# B&R Automation Studio project Panasonic_LinkaPowerCP2_A2021055 (part 33)

#### Main.st - Init, cyclic, exit code
```iecst
PROGRAM _INIT

	//Init parametre serva zdvihu výťahu//
	P4_Vytah.ServoZdvihuVytahu.Parameters.Override:= 100;
	P4_Vytah.PAR.Zdvih_JoggRychlost:= 5;
	P4_Vytah.ServoZdvihuVytahu.Command.TorqueLimitation:= TRUE;
	P4_Vytah.ServoZdvihuVytahu.Parameters.Torque:= 1.0;

END_PROGRAM

PROGRAM _CYCLIC

	//Volanie podprogramov a knižníc//
	IOLinkKomunikacia;

	//Volanie funkcie SequenceControl//
	SequenceControl(SC:= SC_P4_Vytah);

	//Enable serva//
	IF Safety.STAV.P4_ZonaVytahu_AKTIVNA AND NOT P4_Vytah.ServoZdvihuVytahu.Command.ErrReset THEN
		P4_Vytah.ServoZdvihuVytahu.Command.PowerON:= TRUE;
	ELSE
		P4_Vytah.ServoZdvihuVytahu.Command.PowerON:= FALSE;
	END_IF

	//Zaokrúhlenie aktuálnej pozície serva zdvihu//
	ServoZdvihu_AktualPosition_UDINT:= REAL_TO_UDINT(P4_Vytah.ServoZdvihuVytahu.Status.ActPosition);

	//Reset poruchy serva//
	IF EDGEPOS(Safety.STAV.P4_ZonaVytahu_AKTIVNA)THEN
		P4_Vytah.ServoZdvihuVytahu.Command.ErrReset:= TRUE;
	END_IF

	CasResetServo_1.IN:= P4_Vytah.ServoZdvihuVytahu.Command.ErrReset;
	IF CasResetServo_1.Q AND NOT P4_Vytah.ServoZdvihuVytahu.Status.Error THEN
		P4_Vytah.ServoZdvihuVytahu.Command.ErrReset:= FALSE;
	END_IF

	CasResetServo_1.PT:= T#500ms;
	CasResetServo_1();

	//Zhasnutie Bannera//
	IF P4_Vytah.CMD.Banner_LED_OFF THEN
		P4_Vytah.Banner.IN.ModraLED_ON:= FALSE;
		P4_Vytah.Banner.IN.CervenaLED_ON:= FALSE;
		P4_Vytah.Banner.IN.CyanLED_ON:= FALSE;
		P4_Vytah.Banner.IN.ModraRotujucaLED_ON:= FALSE;
		P4_Vytah.Banner.IN.OranzovaLED_ON:= FALSE;
		P4_Vytah.Banner.IN.ZelenaLED_ON:= FALSE;
		P4_Vytah.Banner.IN.ZltaLED_ON:= FALSE;
		P4_Vytah.CMD.Banner_LED_OFF:= FALSE;
	END_IF

	//Reset sekcie //
	IF P4_Vytah.Reset THEN
		SC_P4_Vytah.Step:= 0;
		P4_Vytah.ServoZdvihuVytahu.Command.ErrReset:= TRUE;
		P4_Vytah.Reset:= FALSE;
	ELSIF NOT Safety.STAV.Linka_ZonaCS_AKTIVNA THEN
		SC_P4_Vytah.Step:= 0;
	END_IF

	CASE SC_P4_Vytah.Step OF

		0:
			SC_P4_Vytah.StepName:='0 - Nulovanie';
			P4_Vytah.Automat:= FALSE;
			P4_Vytah.KoniecCyklu:= FALSE;
			P4_Vytah.Manual:= FALSE;
			P4_Vytah.STAV.PoINIT:= FALSE;
			P4_Vytah.ServoZdvihuVytahu.Command.JogNeg:= FALSE;
			P4_Vytah.ServoZdvihuVytahu.Command.JogPos:= FALSE;
			P4_Vytah.ServoZdvihuVytahu.Command.MoveAdditive:= FALSE;
			P4_Vytah.ServoZdvihuVytahu.Command.MovePosition:= FALSE;
			IF NOT P4_Vytah.ServoZdvihuVytahu.Status.StandStill THEN
				P4_Vytah.ServoZdvihuVytahu.Command.Stop:= TRUE;
			END_IF
			P4_Vytah.OUT.DopravnikChod_VPRED:= FALSE;
			P4_Vytah.OUT.DopravnikChod_VZAD:= FALSE;
			P4_Vytah.CMD.Banner_LED_OFF:= TRUE;
			P4_Vytah.RFID_hlava.PrecitajChipRFID:= FALSE;
			TRCB_P4_Vytah_ST10.CMD.VyziadajStavPaletky_TYP1:= FALSE;
			TRCB_P4_Vytah_ST10.CMD.PriradQRkodFiltra_TYP3:= FALSE;
			TRCB_P4_Vytah_ST10.CMD.OdosliStavPaletky_TYP2:= FALSE;
			TRCB_P4_Vytah_ST10.CMD.VyziadajStavPanatrace_TYP4:= FALSE;
			P4_Vytah.CMD.RR_ChodDopravnika_VPRED:= FALSE;
			P4_Vytah.CMD.RR_ChodDopravnika_VZAD:= FALSE;
			P4_Vytah.CMD.RR_ZdvihVytahu_DOLE:= FALSE;
			P4_Vytah.CMD.RR_ZdvihVytahu_HORE:= FALSE;
			CAM16.CMD.Triger:= FALSE;
			CAM16.STAV.Results_READY:= FALSE;
			FTP_CAM16.CMD.OdosliFotku:= FALSE;
			FTP_CAM16.CMD.VymazFotku:= FALSE;
			P34_Vizu.ZobrazHL1_ST10:= FALSE;
			P34_Vizu.ZobrazHL2_ST10:= FALSE;
			P34_Vizu.ZobrazHL3_ST10:= FALSE;
			P34_Vizu.ZobrazHL4_ST10:= FALSE;
			P34_Vizu.ZobrazHL5_ST10:= FALSE;
			P34_Vizu.ZobrazHL6_ST10:= FALSE;
			P34_Vizu.ZobrazHL7_ST10:= FALSE;
			P34_Vizu.ZobrazHL8_ST10:= FALSE;
			P34_Vizu.ZobrazHL9_ST10:= FALSE;
			P34_Vizu.ZobrazHL10_ST10:= FALSE;
			P4_Vytah_KAM_Result_Ignoruj:= FALSE;
			P4_Vytah_KAM_Result_OK:= FALSE;
			P4_Vytah_KAM_Result_NG:= FALSE;
			P4_Vytah.PAR.IndexFotky:= 0;
			TRCB_P4_Vytah_OpatovnyDopyt:= FALSE;
			TRCB_P4_Vytah_PaletkaNG:= FALSE;
			PocetTrigrovKamery:= 0;
			PocetDopytovNaServer:= 0;
			CisloFotky:= 0;
			TestovaciKus:= FALSE;
			Stav_VlozenaPaletka:= FALSE;
			P4_Vytah_Taktime.IN.START_MeraniaCasu:= FALSE;
			P4_Etiketovacka.STAV.PrebiehaVyvezeniePaletky:= FALSE;
			P4_Vytah.STAV.PrebiehaVyvezeniePaletky:= FALSE;
			P4_Vytah_Taktime.IN.START_MeraniaStratovehoCasu:= FALSE;

			IF Safety.STAV.P4_ZonaVytahu_AKTIVNA AND
				P4_Pracovisko.STAV.HardwareVytahu_OK AND
				NOT P4_Pracovisko.STAV.Porucha_ST6 AND
				(P4_Vytah.ServoZdvihuVytahu.Status.Ready AND P4_Vytah.ServoZdvihuVytahu.Status.StandStill) THEN
				P4_Vytah.ServoZdvihuVytahu.Command.Stop:= FALSE;
				SC_P4_Vytah.ResetStep:= TRUE;
				SC_P4_Vytah.Step:= 1;
			END_IF

		1:
			SC_P4_Vytah.StepName:='1 - Cakam na spustenie vyroby';
			P4_Vytah.KoniecCyklu:= FALSE;
			IF P4_Vytah.Automat THEN
				SC_P4_Vytah.Step:= 2;
			ELSIF P4_Vytah.Manual THEN
				SC_P4_Vytah.Step:= 700;
			END_IF

			//********************************************************Inicializácia****************************************************************************//

		2:
			SC_P4_Vytah.StepName:='2 - Inicializacia - cakam na spustenie inicializacie';
			SC_P4_Vytah.IdleTime.PT:= T#2s;
			SC_P4_Vytah.AlarmTime.PT:= T#5s;

			SC_P4_Vytah.IdleTime.IN:= P4_Dopravniky.STAV.PoINIT;

			P4_Vytah.ServoZdvihuVytahu.Parameters.Acc:= P34_RemPremenne.P4_Vytah_Zdvih_Acc;
			P4_Vytah.ServoZdvihuVytahu.Parameters.Dcc:= P34_RemPremenne.P4_Vytah_Zdvih_Dcc;
			P4_Vytah.ServoZdvihuVytahu.Parameters.Torque:= 1.5;

			IF SC_P4_Vytah.IdleTime.Q THEN
				SC_P4_Vytah.ResetStep:= TRUE;
				SC_P4_Vytah.Step:= 3;
			END_IF

		3:
			SC_P4_Vytah.StepName:='3 - Inicializacia - vymazanie adresara kamery';
			SC_P4_Vytah.IdleTime.PT:= T#4s;
			SC_P4_Vytah.AlarmTime.PT:= T#5s;

			P4_Vytah.Banner.IN.ModraLED_ON:= TRUE;

			IF NOT SC_P4_Vytah.Switch1 THEN
				FTP_CAM16.CMD.VymazFotku:= TRUE;
				SC_P4_Vytah.Switch1:= TRUE;
			END_IF

			IF FTP_CAM16.STATUS.KomunikaciaUkoncena THEN
				P4_Vytah.CMD.Banner_LED_OFF:= TRUE;
				FTP_CAM16.CMD.VymazFotku:= FALSE;
				SC_P4_Vytah.ResetStep:= TRUE;
				SC_P4_Vytah.Step:= 4;
			ELSIF FTP_CAM16.STATUS.KomunikaciaError THEN
				P34_Alarmy[410]:= TRUE;
				P4_Pracovisko.STAV.Porucha_ST6:= TRUE;
			END_IF

		4:
			SC_P4_Vytah.StepName:='4 - Inicializacia - spustam dopravnik vytahu pre navezenie paletky';
			SC_P4_Vytah.IdleTime.PT:= T#500ms;
			SC_P4_Vytah.AlarmTime.PT:= T#7s;

			SC_P4_Vytah.IdleTime.IN:= P4_Vytah.RFID_hlava.PritomnostPaletky;

			IF NOT SC_P4_Vytah.Switch1 THEN
				P4_Vytah.OUT.DopravnikChod_VPRED:= TRUE;
				SC_P4_Vytah.AlarmTime.IN:= TRUE;
				SC_P4_Vytah.Switch1:= TRUE;
			END_IF

			IF SC_P4_Vytah.IdleTime.Q AND NOT P4_Vytah.IN.PrechodDopravnika THEN
				P4_Vytah.OUT.DopravnikChod_VPRED:= FALSE;
				SC_P4_Vytah.ResetStep:= TRUE;
				SC_P4_Vytah.Step:= 13;
			ELSIF SC_P4_Vytah.AlarmTime.Q AND NOT P4_Vytah.RFID_hlava.PritomnostPaletky AND NOT P4_Vytah.IN.PrechodDopravnika THEN
				P4_Vytah.OUT.DopravnikChod_VPRED:= FALSE;
				SC_P4_Vytah.ResetStep:= TRUE;
				SC_P4_Vytah.Step:= 13;
			ELSIF SC_P4_Vytah.IdleTime.Q AND P4_Vytah.IN.PrechodDopravnika THEN
				P34_Alarmy[411]:= TRUE;
				P4_Pracovisko.STAV.Porucha_ST6:= TRUE;
			END_IF

		13:
			SC_P4_Vytah.StepName:='13 - Inicializacia - presuvam vytah do hornej pozicie vyvazania';
			SC_P4_Vytah.IdleTime.PT:= T#1s;
			SC_P4_Vytah.AlarmTime.PT:= T#5s;

			SC_P4_Vytah.IdleTime.IN:= Safety.STAV.P4_Vytah_Bariera_AKTIVNA;
			P34_Vizu.ZobrazHL6_ST10:= NOT Safety.STAV.P4_Vytah_Bariera_AKTIVNA;

			P4_Vytah.ServoZdvihuVytahu.Parameters.Velocity:= P34_RemPremenne.P4_Vytah_RychlostZdvihu/1000;
			P4_Vytah.ServoZdvihuVytahu.Parameters.Position:= P34_RemPremenne.P4_Vytah_PoziciaNakladania;

			P4_Vytah.Banner.IN.OranzovaLED_ON:= Blikac1s;

			IF NOT SC_P4_Vytah.Switch1 AND SC_P4_Vytah.IdleTime.Q THEN
				P4_Vytah.ServoZdvihuVytahu.Command.MovePosition:= TRUE;
				SC_P4_Vytah.Switch1:= TRUE;
			END_IF

			IF EDGEPOS(P4_Vytah.ServoZdvihuVytahu.Status.InPosition) THEN
				P4_Vytah.ServoZdvihuVytahu.Command.MovePosition:= FALSE;
				P4_Vytah.CMD.Banner_LED_OFF:= TRUE;
				P34_Vizu.ZobrazHL6_ST10:= FALSE;
				SC_P4_Vytah.ResetStep:= TRUE;
				SC_P4_Vytah.Step:= 15;
			END_IF

		15:
			SC_P4_Vytah.StepName:='15 - Inicializacia - kontrola pritomnosti paletky';
			SC_P4_Vytah.IdleTime.PT:= T#2s;
			SC_P4_Vytah.AlarmTime.PT:= T#5s;

			IF P4_Vytah.RFID_hlava.PritomnostPaletky THEN
				SC_P4_Vytah.ResetStep:= TRUE;
				SC_P4_Vytah.Step:= 18;
			ELSE
				P4_Vytah.STAV.PoINIT:= TRUE;
				SC_P4_Vytah.ResetStep:= TRUE;
				SC_P4_Vytah.Step:= 100;
			END_IF

		18:
			SC_P4_Vytah.StepName:='18 - Inicializacia -  precitanie cisla paletky';
			SC_P4_Vytah.IdleTime.PT:= T#200ms;
			SC_P4_Vytah.AlarmTime.PT:= T#5s;

			SC_P4_Vytah.IdleTime.IN:= P4_Vytah.RFID_hlava.PritomnostPaletky;

			IF SC_P4_Vytah.IdleTime.Q AND NOT SC_P4_Vytah.Switch1 THEN
				P4_Vytah.RFID_hlava.PrecitajChipRFID:= TRUE;
				i:= 0;
				SC_P4_Vytah.Switch1:= TRUE;
			END_IF

			IF P4_Vytah.RFID_hlava.Stav_CitanieZapis_OK AND P4_Vytah.RFID_hlava.PrecitaneCisloPaletky <> 0 THEN
				i:= P4_Vytah.RFID_hlava.PrecitaneCisloPaletky;
				P4_Vytah.PAR.CisloPaletky:= P4_Vytah.RFID_hlava.PrecitaneCisloPaletky;
				P4_Vytah.RFID_hlava.PrecitajChipRFID:= FALSE;
				SC_P4_Vytah.ResetStep:= TRUE;
				SC_P4_Vytah.Step:= 20;
			END_IF

		20:
			SC_P4_Vytah.StepName:='20 - Inicializacia - priradenie indexu paletky na zaklade precitanej hodnoty';
			SC_P4_Vytah.IdleTime.PT:= T#200ms;
			SC_P4_Vytah.AlarmTime.PT:= T#5s;

			IF i<> 0 THEN
				P4_Vytah.PAR.CisloPaletky_STRING:= USINT_TO_STRING(i);
				Paletka[i].PAR.CisloPaletky:= USINT_TO_STRING(i);
				SC_P4_Vytah.ResetStep:= TRUE;
				SC_P4_Vytah.Step:= 30;
			ELSE
				P34_Alarmy[418]:= TRUE;
				P4_Pracovisko.STAV.Porucha_ST6:= TRUE;
			END_IF

		30:
			SC_P1_StoperSrobovania.StepName:='30 - Inicializacia - kontrola stavu paletky';
			SC_P4_Vytah.IdleTime.PT:= T#200ms;
			SC_P4_Vytah.AlarmTime.PT:= T#5s;

			IF Paletka[i].STAV.StavPaletky = '' THEN
				P4_Vytah.STAV.PoINIT:= TRUE;
				Paletka[i].STAV.StavPaletky:= 'NG';
				SC_P4_Vytah.ResetStep:= TRUE;
				SC_P4_Vytah.Step:= 560;
			ELSIF Paletka[i].STAV.StavPaletky = 'PRECH' THEN
				P4_Vytah.STAV.PoINIT:= TRUE;
				SC_P4_Vytah.ResetStep:= TRUE;
				SC_P4_Vytah.Step:= 130;
			ELSIF Paletka[i].STAV.StavPaletky = 'TEST' THEN
				P4_Vytah.STAV.PoINIT:= TRUE;
				SC_P4_Vytah.ResetStep:= TRUE;
				SC_P4_Vytah.Step:= 130;
			ELSIF Paletka[i].STAV.StavPaletky = 'REV' AND Paletka[i].STAV.CisloRevorkovejStanice = 'ST_10' THEN
				Paletka[i].STAV.StavPaletky:= 'OK';
				SC_P4_Vytah.ResetStep:= TRUE;
				SC_P4_Vytah.Step:= 33;
			ELSIF Paletka[i].STAV.StavPaletky = 'REV' AND Paletka[i].STAV.CisloRevorkovejStanice <> 'ST_10' THEN
				P4_Vytah.STAV.PoINIT:= TRUE;
				SC_P4_Vytah.ResetStep:= TRUE;
				SC_P4_Vytah.Step:= 130;
			ELSIF Paletka[i].STAV.StavPaletky = 'OK' THEN
				SC_P4_Vytah.ResetStep:= TRUE;
				SC_P4_Vytah.Step:= 33;
			ELSIF Paletka[i].STAV.StavPaletky = 'NG' THEN
				P4_Vytah.STAV.PoINIT:= TRUE;
				SC_P4_Vytah.ResetStep:= TRUE;
				SC_P4_Vytah.Step:= 130;
			END_IF

		33:
			SC_P4_Vytah.StepName:='33 - Inicializacia - kontrola uzavretia komunikacie s Panatrace';
			SC_P4_Vytah.IdleTime.PT:= T#5s;
			SC_P4_Vytah.AlarmTime.PT:= T#5s;

			IF Paletka[i].STAV.Komunikacia_DONE THEN
				P4_Vytah.STAV.PoINIT:= TRUE;
				SC_P4_Vytah.ResetStep:= TRUE;
				SC_P4_Vytah.Step:= 130;
			ELSE
				P4_Vytah.STAV.PoINIT:= TRUE;
				SC_P4_Vytah.ResetStep:= TRUE;
				SC_P4_Vytah.Step:= 111;
			END_IF

			//********************************************************Automatický režim****************************************************************************//

		100:
			SC_P4_Vytah.StepName:='100 - Automaticky Rezim - cakam na navezenie paletky na vytah z vrchneho dopravnika';
			SC_P4_Vytah.IdleTime.PT:= T#200ms;
			SC_P4_Vytah.AlarmTime.PT:= T#5s;

			P4_Vytah.ServoZdvihuVytahu.Parameters.Acc:= P34_RemPremenne.P4_Vytah_Zdvih_Acc;
			P4_Vytah.ServoZdvihuVytahu.Parameters.Dcc:= P34_RemPremenne.P4_Vytah_Zdvih_Dcc;
			P4_Vytah.ServoZdvihuVytahu.Parameters.Torque:= 1.5;

			IF P4_Vytah.KoniecCyklu AND NOT P4_Etiketovacka.Automat THEN
				SC_P4_Vytah.ResetStep:= TRUE;
				SC_P4_Vytah.Step:= 0;
			ELSIF SC_P4_Etiketovacka.Step = 561 AND NOT P4_Vytah.RFID_hlava.PritomnostPaletky AND NOT P4_Vytah.IN.PrechodDopravnika THEN
				Stav_VlozenaPaletka:= FALSE;
				SC_P4_Vytah.ResetStep:= TRUE;
				SC_P4_Vytah.Step:= 101;
			ELSIF P4_Vytah.RFID_hlava.PritomnostPaletky THEN
				P4_Etiketovacka.STAV.PrebiehaVyvezeniePaletky:= FALSE;
				Stav_VlozenaPaletka:= TRUE;
				SC_P4_Vytah.ResetStep:= TRUE;
				SC_P4_Vytah.Step:= 105;
			END_IF

		101:
			SC_P4_Vytah.StepName:='101 - Automaticky Rezim - navazam paletku na dopravnik vytahu';
			SC_P4_Vytah.IdleTime.PT:= T#200ms;
			SC_P4_Vytah.AlarmTime.PT:= T#20s;

			SC_P4_Vytah.IdleTime.IN:= P4_Vytah.RFID_hlava.PritomnostPaletky;

			IF NOT SC_P4_Vytah.Switch2 AND P4_Vytah.RFID_hlava.PritomnostPaletky THEN
				P4_Vytah_Taktime.IN.START_MeraniaCasu:= TRUE;
				P4_Vytah_Taktime.IN.ZAPIS_MeraniaCasu:= TRUE;
				P4_Vytah_Taktime.IN.ZAPIS_StratovyCas:= TRUE;
				Buffer_14.Hodnota:= P4_Vytah_Taktime.OUT.StratoveSekundy;
				Buffer_14.ZapisHodnotu:= TRUE;
				SC_P4_Vytah.Switch2:= TRUE;
			END_IF

			IF NOT SC_P4_Vytah.Switch1 THEN
				P4_Vytah.OUT.DopravnikChod_VPRED:= TRUE;
				SC_P4_Vytah.AlarmTime.IN:= TRUE;
				SC_P4_Vytah.Switch1:= TRUE;
			END_IF

			IF SC_P4_Vytah.IdleTime.Q THEN
				P4_Etiketovacka.STAV.PrebiehaVyvezeniePaletky:= FALSE;
				P4_Vytah.OUT.DopravnikChod_VPRED:= FALSE;
				SC_P4_Vytah.ResetStep:= TRUE;
				SC_P4_Vytah.Step:= 105;
			ELSIF SC_P4_Vytah.AlarmTime.Q THEN
				P34_Alarmy[416]:= TRUE;
				P4_Pracovisko.STAV.Porucha_ST6:= TRUE;
			END_IF

		105:
			SC_P4_Vytah.StepName:='105 - Automaticky Rezim - precitanie cisla paletky';
			SC_P4_Vytah.IdleTime.PT:= T#500ms;
			SC_P4_Vytah.AlarmTime.PT:= T#5s;
			SC_P4_Vytah.IdleTime.IN:= TRUE;

			IF NOT SC_P4_Vytah.Switch1 THEN
				i:= 0;
				P4_Vytah.RFID_hlava.PrecitajChipRFID:= TRUE;
				SC_P4_Vytah.Switch1:= TRUE;
			END_IF

			IF P4_Vytah.RFID_hlava.Stav_CitanieZapis_OK AND P4_Vytah.RFID_hlava.PrecitaneCisloPaletky <> 0 THEN
				i:= P4_Vytah.RFID_hlava.PrecitaneCisloPaletky;
				P4_Vytah.PAR.CisloPaletky:= P4_Vytah.RFID_hlava.PrecitaneCisloPaletky;
				P4_Vytah.RFID_hlava.PrecitajChipRFID:= FALSE;
				SC_P4_Vytah.ResetStep:= TRUE;
				SC_P4_Vytah.Step:= 108;
			END_IF

		108:
			SC_P4_Vytah.StepName:='108 - Automaticky Rezim - kontrola a priradenie indexu paletky na zaklade precitanej hodnoty';
			SC_P4_Vytah.IdleTime.PT:= T#200ms;
			SC_P4_Vytah.AlarmTime.PT:= T#5s;

			IF i<> 0 THEN
				P4_Vytah.PAR.CisloPaletky_STRING:= USINT_TO_STRING(i);
				Paletka[i].PAR.CisloPaletky:= USINT_TO_STRING(i);
				SC_P4_Vytah.ResetStep:= TRUE;
				SC_P4_Vytah.Step:= 110;
			ELSE
				P34_Alarmy[418]:= TRUE;
				P4_Pracovisko.STAV.Porucha_ST6:= TRUE;
			END_IF

		110:
			SC_P4_Vytah.StepName:='110 - Automaticky Rezim - kontrola stavu paletky';
			SC_P4_Vytah.IdleTime.PT:= T#200ms;
			SC_P4_Vytah.AlarmTime.PT:= T#5s;

			IF Paletka[i].STAV.StavPaletky = '' THEN
				Paletka[i].STAV.StavPaletky:= 'NG';
				SC_P4_Vytah.ResetStep:= TRUE;
				SC_P4_Vytah.Step:= 560;
			ELSIF Paletka[i].STAV.StavPaletky = 'PRECH' THEN
				SC_P4_Vytah.ResetStep:= TRUE;
				SC_P4_Vytah.Step:= 130;
			ELSIF Paletka[i].STAV.StavPaletky = 'TEST' THEN
				SC_P4_Vytah.ResetStep:= TRUE;
				SC_P4_Vytah.Step:= 130;
			ELSIF Paletka[i].STAV.StavPaletky = 'REV' AND Paletka[i].STAV.CisloRevorkovejStanice = 'ST_10' THEN
				Paletka[i].STAV.StavPaletky:= 'OK';
				SC_P4_Vytah.ResetStep:= TRUE;
				SC_P4_Vytah.Step:= 111;
			ELSIF Paletka[i].STAV.StavPaletky = 'REV' AND Paletka[i].STAV.CisloRevorkovejStanice <> 'ST_10' THEN
				SC_P4_Vytah.ResetStep:= TRUE;
				SC_P4_Vytah.Step:= 130;
			ELSIF Paletka[i].STAV.StavPaletky = 'OK' THEN
				SC_P4_Vytah.ResetStep:= TRUE;
				SC_P4_Vytah.Step:= 111;
			ELSIF Paletka[i].STAV.StavPaletky = 'NG' THEN
				SC_P4_Vytah.ResetStep:= TRUE;
				SC_P4_Vytah.Step:= 130;
			END_IF

		111:
			SC_P4_Vytah.StepName:='111 - Automaticky Rezim - kontrola prihlasenia operatora';
			SC_P4_Vytah.IdleTime.PT:= T#1s;
			SC_P4_Vytah.AlarmTime.PT:= T#5s;

			IF P34_UzivatelPrihlaseny THEN
				Paletka[i].PAR.ID_Operatora:= 'E2';//UsersVizu.CisloPrihlasenejKarty_Panel3;
				P34_Vizu.ZobrazHL7_ST10:= FALSE;
				P4_Vytah.CMD.Banner_LED_OFF:= FALSE;
				SC_P4_Vytah.ResetStep:= TRUE;
				SC_P4_Vytah.Step:= 112;
			ELSE
				P4_Vytah.Banner.IN.CyanLED_ON:= Blikac500ms;
				P34_Vizu.ZobrazHL7_ST10:= TRUE;
				Paletka[i].PAR.ID_Operatora:= '';
			END_IF

		112:
			SC_P4_Vytah.StepName:='112 - Automaticky Rezim - vyziadanie stavu komunikacie zo serverom';
			SC_P4_Vytah.IdleTime.PT:= T#200ms;
			SC_P4_Vytah.AlarmTime.PT:= T#10s;

			P4_Vytah.Banner.IN.ModraRotujucaLED_ON:= TRUE;

			IF Linka.KOM_Panatrace_OFF THEN
				CAM16.STAV.Results_READY:= FALSE;
				CAM16.STAV.OldRunCounter:= CAM16.STAV.RunCounter;
				P4_Vytah.CMD.Banner_LED_OFF:= TRUE;
				SC_P4_Vytah.ResetStep:= TRUE;
				SC_P4_Vytah.Step:= 118;
			ELSIF NOT SC_P4_Vytah.Switch1 AND TRCB_P4_Vytah_ST10.STATUS.KOM_READY THEN
				TRCB_P4_Vytah_ST10.CMD.VyziadajStavPanatrace_TYP4:= TRUE;
				(*P4_Vytah_Taktime.IN.START_MeraniaStratovehoCasu:= TRUE;*)
				SC_P4_Vytah.Switch1:= TRUE;
			END_IF

			IF TRCB_P4_Vytah_ST10.STATUS.KomunikaciaUkoncena THEN
				P4_Vytah.CMD.Banner_LED_OFF:= TRUE;
				TRCB_P4_Vytah_ST10.CMD.VyziadajStavPanatrace_TYP4:= FALSE;
				P4_Vytah_Taktime.IN.START_MeraniaStratovehoCasu:= FALSE;
				SC_P4_Vytah.ResetStep:= TRUE;
				SC_P4_Vytah.Step:= 113;
			ELSIF TRCB_P4_Vytah_ST10.STATUS.KomunikaciaError THEN
				P4_Vytah.CMD.Banner_LED_OFF:= TRUE;
				TRCB_P4_Vytah_ST10.CMD.VyziadajStavPanatrace_TYP4:= FALSE;
				P4_Vytah_Taktime.IN.START_MeraniaStratovehoCasu:= FALSE;
				SC_P4_Vytah.ResetStep:= TRUE;
				SC_P4_Vytah.Step:= 114;
			END_IF

		113:
			SC_P4_Vytah.StepName:='113 - Automaticky Rezim - kontrola odpovede servera';
			SC_P4_Vytah.IdleTime.PT:= T#200ms;
			SC_P4_Vytah.AlarmTime.PT:= T#5s;

			IF NOT TRCB_P4_Vytah_ST10.STATUS.KomunikaciaUkoncena THEN
				IF TRCB_P4_Vytah_ST10.OUTPUTS.DruhCinnostiNaPaletke = '0;Generating' THEN
					SC_P4_Vytah.ResetStep:= TRUE;
					SC_P4_Vytah.Step:= 114;
				ELSIF TRCB_P4_Vytah_ST10.OUTPUTS.DruhCinnostiNaPaletke = '1;Request' THEN
					SC_P4_Vytah.ResetStep:= TRUE;
					SC_P4_Vytah.Step:= 115;
				ELSIF TRCB_P4_Vytah_ST10.OUTPUTS.DruhCinnostiNaPaletke = '2;Report' THEN
					CAM16.STAV.OldRunCounter:= CAM16.STAV.RunCounter;
					CAM16.STAV.Results_READY:= FALSE;
					SC_P4_Vytah.ResetStep:= TRUE;
					SC_P4_Vytah.Step:= 118;
				ELSIF TRCB_P4_Vytah_ST10.OUTPUTS.DruhCinnostiNaPaletke = '3;Wedding' THEN
					SC_P4_Vytah.ResetStep:= TRUE;
					SC_P4_Vytah.Step:= 114;
				ELSIF TRCB_P4_Vytah_ST10.OUTPUTS.DruhCinnostiNaPaletke = '4;Status' THEN
					SC_P4_Vytah.ResetStep:= TRUE;
					SC_P4_Vytah.Step:= 114;
				ELSIF TRCB_P4_Vytah_ST10.OUTPUTS.DruhCinnostiNaPaletke = '5;' THEN
					SC_P4_Vytah.ResetStep:= TRUE;
					SC_P4_Vytah.Step:= 114;
				ELSE
					SC_P4_Vytah.ResetStep:= TRUE;
					SC_P4_Vytah.Step:= 114;
				END_IF
			END_IF

		114:
			SC_P4_Vytah.StepName:='114 - Automaticky Rezim - rozhodnutie obsluhy po chybe komunikacie s Panatrace';
			SC_P4_Vytah.IdleTime.PT:= T#200ms;
			SC_P4_Vytah.AlarmTime.PT:= T#5s;

			P34_Vizu.ZobrazHL10_ST10:= TRUE;

			IF TRCB_P4_Vytah_OpatovnyDopyt THEN
				TRCB_P4_Vytah_OpatovnyDopyt:= FALSE;
				P34_Vizu.ZobrazHL10_ST10:= FALSE;
				SC_P4_Vytah.ResetStep:= TRUE;
				SC_P4_Vytah.Step:= 112;
			ELSIF TRCB_P4_Vytah_PaletkaNG THEN
				TRCB_P4_Vytah_PaletkaNG:= FALSE;
				P34_Vizu.ZobrazHL10_ST10:= FALSE;
				Paletka[i].STAV.StavPaletky := 'NG';
				SC_P4_Vytah.ResetStep:= TRUE;
				SC_P4_Vytah.Step:= 130;
			END_IF

		115:
			SC_P4_Vytah.StepName:='115 - Automaticky Rezim - vyziadanie stavu paletky zo servera';
			SC_P4_Vytah.IdleTime.PT:= T#200ms;
			SC_P4_Vytah.AlarmTime.PT:= T#5s;
			SC_P4_Vytah.IdleTime.IN:= TRUE;

			IF NOT SC_P4_Vytah.Switch1 AND TRCB_P4_Vytah_ST10.STATUS.KOM_READY THEN
				TRCB_P4_Vytah_ST10.CMD.VyziadajStavPaletky_TYP1:= TRUE;
				(*P4_Vytah_Taktime.IN.START_MeraniaStratovehoCasu:= TRUE;*)
				SC_P4_Vytah.Switch1:= TRUE;
			END_IF

			IF TRCB_P4_Vytah_ST10.STATUS.KomunikaciaUkoncena THEN
				P4_Vytah.CMD.Banner_LED_OFF:= TRUE;
				TRCB_P4_Vytah_ST10.CMD.VyziadajStavPaletky_TYP1:= FALSE;
				P4_Vytah_Taktime.IN.START_MeraniaStratovehoCasu:= FALSE;
				SC_P4_Vytah.ResetStep:= TRUE;
				SC_P4_Vytah.Step:= 116;
			ELSIF TRCB_P4_Vytah_ST10.STATUS.KomunikaciaError THEN
				P4_Vytah.CMD.Banner_LED_OFF:= TRUE;
				TRCB_P4_Vytah_ST10.CMD.VyziadajStavPaletky_TYP1:= FALSE;
				P4_Vytah_Taktime.IN.START_MeraniaStratovehoCasu:= FALSE;
				SC_P4_Vytah.ResetStep:= TRUE;
				SC_P4_Vytah.Step:= 114;
			END_IF

		116:
			SC_P4_Vytah.StepName:='116 - Automaticky Rezim - kontrola odpovede servera';
			SC_P4_Vytah.IdleTime.PT:= T#200ms;
			SC_P4_Vytah.AlarmTime.PT:= T#5s;

			IF NOT TRCB_P4_Vytah_ST10.STATUS.KomunikaciaUkoncena THEN
				IF TRCB_P4_Vytah_ST10.OUTPUTS.PovolenieCinnostiNaPaletke = 'OK' THEN
					CAM16.STAV.Results_READY:= FALSE;
					CAM16.STAV.OldRunCounter:= CAM16.STAV.RunCounter;
					SC_P4_Vytah.ResetStep:= TRUE;
					SC_P4_Vytah.Step:= 118;
				ELSIF TRCB_P4_Vytah_ST10.OUTPUTS.PovolenieCinnostiNaPaletke = 'NG' THEN
					SC_P4_Vytah.ResetStep:= TRUE;
					SC_P4_Vytah.Step:= 117;
				END_IF
			END_IF

		117:
			SC_P4_Vytah.StepName:='117 - Automaticky Rezim - rozhodnutie obsluhy po odpovedi panatrace NG';
			SC_P4_Vytah.IdleTime.PT:= T#200ms;
			SC_P4_Vytah.AlarmTime.PT:= T#5s;

			P34_Vizu.ZobrazHL9_ST10:= TRUE;

			IF TRCB_P4_Vytah_OpatovnyDopyt THEN
				TRCB_P4_Vytah_OpatovnyDopyt:= FALSE;
				P34_Vizu.ZobrazHL9_ST10:= FALSE;
				SC_P4_Vytah.ResetStep:= TRUE;
				SC_P4_Vytah.Step:= 112;
			ELSIF TRCB_P4_Vytah_PaletkaNG THEN
				TRCB_P4_Vytah_PaletkaNG:= FALSE;
				P34_Vizu.ZobrazHL9_ST10:= FALSE;
				Paletka[i].STAV.StavPaletky := 'NG';
				SC_P4_Vytah.ResetStep:= TRUE;
				SC_P4_Vytah.Step:= 130;
			END_IF

		118:
			SC_P4_Vytah.StepName:='118 - Automaticky Rezim - kamerova kontrola paletky CAM16';//CAM 16
			SC_P4_Vytah.IdleTime.PT:= T#5s;
			SC_P4_Vytah.AlarmTime.PT:= T#5s;

			P4_Vytah.Banner.IN.ModraLED_ON:= TRUE;

			IF NOT SC_P4_Vytah.Switch1 AND CAM16.STAV.Command_READY THEN
				CAM16.CMD.Triger:= TRUE;
				SC_P4_Vytah.IdleTime.IN:= TRUE;
				SC_P4_Vytah.Switch1:= TRUE;
			END_IF

			IF CAM16.STAV.Results_READY AND CAM16.STAV.Command_AKCEPTOVANY AND CAM16.STAV.OldRunCounter <> CAM16.STAV.RunCounter THEN
				PocetTrigrovKamery:= 0;
				CAM16.STAV.Results_READY:= FALSE;
				CAM16.STAV.OldRunCounter:= CAM16.STAV.RunCounter;
				CAM16.CMD.Triger:= FALSE;
				P4_Vytah.CMD.Banner_LED_OFF:= TRUE;
				SC_P4_Vytah.ResetStep:= TRUE;
				SC_P4_Vytah.Step:= 120;
			ELSIF SC_P4_Vytah.IdleTime.Q AND PocetTrigrovKamery < 5 THEN
				PocetTrigrovKamery:= PocetTrigrovKamery + 1;
				CAM16.CMD.Triger:= FALSE;
				CAM16.STAV.Results_READY:= FALSE;
				CAM16.STAV.OldRunCounter:= CAM16.STAV.RunCounter;
				P4_Vytah.CMD.Banner_LED_OFF:= TRUE;
				SC_P4_Vytah.ResetStep:= TRUE;
				SC_P4_Vytah.Step:= 119;
			ELSIF SC_P4_Vytah.IdleTime.Q AND PocetTrigrovKamery >= 5 THEN
				P34_Alarmy[455]:= TRUE;
				P4_Pracovisko.STAV.Porucha_ST6:= TRUE;
			END_IF

		119:
			SC_P4_Vytah.StepName:='119 - Automaticky Rezim - cakam na opatovny triger kamery CAM16';
			SC_P4_Vytah.IdleTime.PT:= T#1s;
			SC_P4_Vytah.AlarmTime.PT:= T#5s;

			SC_P4_Vytah.IdleTime.IN:= TRUE;

			IF SC_P4_Vytah.IdleTime.Q THEN
				SC_P4_Vytah.ResetStep:= TRUE;
				SC_P4_Vytah.Step:= 118;
			END_IF

		120:
			SC_P4_Vytah.StepName:='120 - Automaticky Rezim - vysledok kamerovej kontroly kamery CAM16';
			SC_P4_Vytah.IdleTime.PT:= T#1s;
			SC_P4_Vytah.AlarmTime.PT:= T#5s;

			IF Linka.P4_Kamery_OFF THEN
				CAM16.CMD.Triger:= FALSE;
				CAM16.PAR.ResultFotky:= 'PASS';
				SC_P4_Vytah.ResetStep:= TRUE;
				SC_P4_Vytah.Step:= 121;
			ELSIF NOT CAM16.STAV.BUSY THEN
				CAM16.CMD.Triger:= FALSE;
				IF Linka.PAR.ZvolenyModel = '4F' THEN
					CAM16.PAR.ResultFotky:= 'PASS';
					SC_P4_Vytah.ResetStep:= TRUE;
					SC_P4_Vytah.Step:= 121;
				ELSIF Linka.PAR.ZvolenyModel = '5F' THEN
					CAM16.PAR.ResultFotky:= 'PASS';
					SC_P4_Vytah.ResetStep:= TRUE;
					SC_P4_Vytah.Step:= 121;
				ELSIF Linka.PAR.ZvolenyModel = '5H' THEN
					CAM16.PAR.ResultFotky:= 'PASS';
					SC_P4_Vytah.ResetStep:= TRUE;
					SC_P4_Vytah.Step:= 121;
				END_IF
			END_IF

		121:
			SC_P4_Vytah.StepName:='121 - Automaticky Rezim - kontrola vysledku kamery';
			SC_P4_Vytah.IdleTime.PT:= T#1s;
			SC_P4_Vytah.AlarmTime.PT:= T#5s;

			IF CAM16.PAR.ResultFotky = 'PASS' THEN
				SC_P4_Vytah.ResetStep:= TRUE;
				SC_P4_Vytah.Step:= 122;
			ELSIF CAM16.PAR.ResultFotky = 'FAIL' THEN
				P34_Vizu.ZobrazHL8_ST10:= TRUE;
				IF P4_Vytah_KAM_Result_OK THEN
					P4_Vytah_KAM_Result_OK:= FALSE;
					P34_Vizu.ZobrazHL8_ST10:= FALSE;
					CAM16.PAR.ResultFotky:= 'PASS';
					SC_P4_Vytah.ResetStep:= TRUE;
					SC_P4_Vytah.Step:= 122;
				ELSIF P4_Vytah_KAM_Result_NG THEN
					P4_Vytah_KAM_Result_NG:= FALSE;
					Paletka[i].PAR.StavPowerCP:= 'FAIL';
					P34_Vizu.ZobrazHL8_ST10:= FALSE;
					SC_P4_Vytah.ResetStep:= TRUE;
					SC_P4_Vytah.Step:= 122;
				END_IF
			END_IF

		122:
			SC_P4_Vytah.StepName:='122 - Automaticky Rezim - odoslanie fotky CAM16 na server Panasonic';
			SC_P4_Vytah.IdleTime.PT:= T#1s;
			SC_P4_Vytah.AlarmTime.PT:= T#5s;
			SC_P4_Vytah.IdleTime.IN:= TRUE;

			P4_Vytah.Banner.IN.ModraRotujucaLED_ON:= TRUE;

			IF Linka.KOM_FTP_OFF THEN
				P4_Vytah.CMD.Banner_LED_OFF:= TRUE;
				SC_P4_Vytah.ResetStep:= TRUE;
				SC_P4_Vytah.Step:= 123;
			ELSIF NOT SC_P4_Vytah.Switch1 THEN
				FTP_CAM16.INPUTS.QRkodPowerCP:= Paletka[i].PAR.QRkodPowerCP;
				CisloFotky:= CisloFotky + 1;
				FTP_CAM16.INPUTS.IndexFotky:= USINT_TO_STRING(CisloFotky);
				FTP_CAM16.INPUTS.Result:= CAM11.PAR.ResultFotky;
				Reports.Kamery.P4_CAM16_KontrolaPaletky:= CAM11.PAR.ResultFotky;
				FTP_CAM16.CMD.OdosliFotku:= TRUE;
				P4_Vytah_Taktime.IN.START_MeraniaStratovehoCasu:= TRUE;
				SC_P4_Vytah.Switch1:= TRUE;
			END_IF

			IF FTP_CAM16.STATUS.KomunikaciaUkoncena THEN
				P4_Vytah.CMD.Banner_LED_OFF:= TRUE;
				FTP_CAM16.CMD.OdosliFotku:= FALSE;
				P4_Vytah_Taktime.IN.START_MeraniaStratovehoCasu:= FALSE;
				Paletka[i].STAV.OdoslanieFotiek_DONE:= TRUE;
				SC_P4_Vytah.ResetStep:= TRUE;
				SC_P4_Vytah.Step:= 123;
			ELSIF FTP_CAM6.STATUS.KomunikaciaError THEN
				P34_Alarmy[413]:= TRUE;
				P4_Pracovisko.STAV.Porucha_ST6:= TRUE;
			END_IF

		123:
			SC_P4_Vytah.StepName:='123 - Automaticky Rezim - odoslanie stavu paletky na server';
			SC_P4_Vytah.IdleTime.PT:= T#500ms;
			SC_P4_Vytah.AlarmTime.PT:= T#5s;
			SC_P4_Vytah.IdleTime.IN:= TRUE;

			P4_Vytah.Banner.IN.ModraRotujucaLED_ON:= TRUE;

			IF Linka.KOM_Panatrace_OFF THEN
				P4_Vytah.CMD.Banner_LED_OFF:= TRUE;
				SC_P4_Vytah.ResetStep:= TRUE;
				SC_P4_Vytah.Step:= 130;
			ELSIF NOT SC_P4_Vytah.Switch1 AND TRCB_P4_Vytah_ST10.STATUS.KOM_READY THEN
				TRCB_P4_Vytah_ST10.CMD.OdosliStavPaletky_TYP2:= TRUE;
				(*P4_Vytah_Taktime.IN.START_MeraniaStratovehoCasu:= TRUE;*)
				SC_P4_Vytah.Switch1:= TRUE;
			END_IF

			IF TRCB_P4_Vytah_ST10.STATUS.KomunikaciaUkoncena THEN
				P4_Vytah.CMD.Banner_LED_OFF:= TRUE;
				TRCB_P4_Vytah_ST10.CMD.OdosliStavPaletky_TYP2:= FALSE;
				P4_Vytah_Taktime.IN.START_MeraniaStratovehoCasu:= FALSE;
				SC_P4_Vytah.ResetStep:= TRUE;
				SC_P4_Vytah.Step:= 124;
			ELSIF TRCB_P4_Vytah_ST10.STATUS.KomunikaciaError THEN
				TRCB_P4_Vytah_ST10.CMD.OdosliStavPaletky_TYP2:= FALSE;
				P4_Vytah_Taktime.IN.START_MeraniaStratovehoCasu:= FALSE;
				SC_P4_Vytah.ResetStep:= TRUE;
				SC_P4_Vytah.Step:= 127;
			END_IF

		124:
			SC_P4_Vytah.StepName:='124 - Automaticky Rezim - kontrola odpovede servera';
			SC_P4_Vytah.IdleTime.PT:= T#200ms;
			SC_P4_Vytah.AlarmTime.PT:= T#5s;

			IF NOT TRCB_P4_Vytah_ST10.STATUS.KomunikaciaUkoncena THEN
				Paletka[i].STAV.Komunikacia_DONE:= TRUE;
				IF TRCB_P4_Vytah_ST10.OUTPUTS.PovolenieCinnostiNaPaletke = 'OK' THEN
					SC_P4_Vytah.ResetStep:= TRUE;
					SC_P4_Vytah.Step:= 130;
				ELSIF TRCB_P4_Vytah_ST10.OUTPUTS.PovolenieCinnostiNaPaletke = 'NG' THEN
					SC_P4_Vytah.ResetStep:= TRUE;
					SC_P4_Vytah.Step:= 130;
				END_IF
			END_IF

		125:
			SC_P4_Vytah.StepName:='125 - Automaticky Rezim - vyziadanie stavu komunikacie zo serverom';
			SC_P4_Vytah.IdleTime.PT:= T#200ms;
			SC_P4_Vytah.AlarmTime.PT:= T#10s;

			P4_Vytah.Banner.IN.ModraRotujucaLED_ON:= TRUE;

			IF NOT SC_P4_Vytah.Switch1 AND TRCB_P4_Vytah_ST10.STATUS.KOM_READY THEN
				TRCB_P4_Vytah_ST10.CMD.VyziadajStavPanatrace_TYP4:= TRUE;
				SC_P4_Vytah.Switch1:= TRUE;
			END_IF

			IF TRCB_P4_Vytah_ST10.STATUS.KomunikaciaUkoncena THEN
				TRCB_P4_Vytah_ST10.CMD.VyziadajStavPanatrace_TYP4:= FALSE;
				SC_P4_Vytah.ResetStep:= TRUE;
				SC_P4_Vytah.Step:= 126;
			ELSIF TRCB_P4_Vytah_ST10.STATUS.KomunikaciaError THEN
				TRCB_P4_Vytah_ST10.CMD.VyziadajStavPanatrace_TYP4:= FALSE;
				SC_P4_Vytah.ResetStep:= TRUE;
				SC_P4_Vytah.Step:= 127;
			END_IF

		126:
			SC_P4_Vytah.StepName:='126 - Automaticky Rezim - kontrola odpovede servera';
			SC_P4_Vytah.IdleTime.PT:= T#200ms;
			SC_P4_Vytah.AlarmTime.PT:= T#5s;

			IF NOT TRCB_P4_Vytah_ST10.STATUS.KomunikaciaUkoncena THEN
				IF TRCB_P4_Vytah_ST10.OUTPUTS.DruhCinnostiNaPaletke = '0;Generating' THEN
					SC_P4_Vytah.ResetStep:= TRUE;
					SC_P4_Vytah.Step:= 127;
				ELSIF TRCB_P4_Vytah_ST10.OUTPUTS.DruhCinnostiNaPaletke = '1;Request' THEN
					SC_P4_Vytah.ResetStep:= TRUE;
					SC_P4_Vytah.Step:= 127;
				ELSIF TRCB_P4_Vytah_ST10.OUTPUTS.DruhCinnostiNaPaletke = '2;Report' THEN
					SC_P4_Vytah.ResetStep:= TRUE;
					SC_P4_Vytah.Step:= 123;
				ELSIF TRCB_P4_Vytah_ST10.OUTPUTS.DruhCinnostiNaPaletke = '3;Wedding' THEN
					SC_P4_Vytah.ResetStep:= TRUE;
					SC_P4_Vytah.Step:= 127;
				ELSIF TRCB_P4_Vytah_ST10.OUTPUTS.DruhCinnostiNaPaletke = '4;Status' THEN
					SC_P4_Vytah.ResetStep:= TRUE;
					SC_P4_Vytah.Step:= 127;
				ELSIF TRCB_P4_Vytah_ST10.OUTPUTS.DruhCinnostiNaPaletke = '5;' THEN
					SC_P4_Vytah.ResetStep:= TRUE;
					SC_P4_Vytah.Step:= 127;
				ELSE
					SC_P4_Vytah.ResetStep:= TRUE;
					SC_P4_Vytah.Step:= 127;
				END_IF
			END_IF

		127:
			SC_P4_Vytah.StepName:='127 - Automaticky Rezim - rozhodnutie obsluhy po chybe komunikacie s Panatrace';
			SC_P4_Vytah.IdleTime.PT:= T#200ms;
			SC_P4_Vytah.AlarmTime.PT:= T#5s;

			P34_Vizu.ZobrazHL10_ST10:= TRUE;

			IF TRCB_P4_Vytah_OpatovnyDopyt THEN
				TRCB_P4_Vytah_OpatovnyDopyt:= FALSE;
				P34_Vizu.ZobrazHL10_ST10:= FALSE;
				SC_P4_Vytah.ResetStep:= TRUE;
				SC_P4_Vytah.Step:= 125;
			ELSIF TRCB_P4_Vytah_PaletkaNG THEN
				TRCB_P4_Vytah_PaletkaNG:= FALSE;
				P34_Vizu.ZobrazHL10_ST10:= FALSE;
				Paletka[i].STAV.StavPaletky := 'NG';
				SC_P4_Vytah.ResetStep:= TRUE;
				SC_P4_Vytah.Step:= 130;
			END_IF

		130:
			SC_P4_Vytah.StepName:='130 - Automaticky Rezim - cakam na spustenie kamerovej kontroly paletky';
			SC_P4_Vytah.IdleTime.PT:= T#500ms;
			SC_P4_Vytah.AlarmTime.PT:= T#20s;

			IF Paletka[i].STAV.StavPaletky = 'NG' THEN
				P4_Vytah.Banner.IN.CervenaLED_ON:= P4_Vytah.RFID_hlava.PritomnostPaletky;
			ELSE
				P4_Vytah.Banner.IN.ZelenaLED_ON:= P4_Vytah.RFID_hlava.PritomnostPaletky;
			END_IF

			IF P4_Vytah.KoniecCyklu THEN
				SC_P4_Vytah.ResetStep:= TRUE;
				SC_P4_Vytah.Step:= 0;
			ELSIF NOT P4_SpodnyStoper.IN.ZaplnenieDopravnika AND P4_Vytah.RFID_hlava.PritomnostPaletky AND Safety.STAV.P4_Vytah_Bariera_AKTIVNA AND P4_Vytah.Banner.OUT.Stlaceny  THEN
				P4_Vytah.CMD.Banner_LED_OFF:= TRUE;
				CAM16.STAV.Results_READY:= FALSE;
				CAM16.STAV.OldRunCounter:= CAM16.STAV.RunCounter;
				SC_P4_Vytah.ResetStep:= TRUE;
				SC_P4_Vytah.Step:= 133;
			ELSIF NOT P4_Vytah.RFID_hlava.PritomnostPaletky THEN
				P4_Vytah.CMD.Banner_LED_OFF:= TRUE;
				SC_P4_Vytah.ResetStep:= TRUE;
				SC_P4_Vytah.Step:= 100;
			END_IF

		133:
			SC_P4_Vytah.StepName:='133 - Automaticky Rezim - kamerova kontrola paletky CAM16';//CAM 16//
			SC_P4_Vytah.IdleTime.PT:= T#5s;
			SC_P4_Vytah.AlarmTime.PT:= T#10s;

			P4_Vytah.Banner.IN.ModraLED_ON:= TRUE;

			IF NOT SC_P4_Vytah.Switch1 AND CAM16.STAV.Command_READY THEN
				CAM16.CMD.Triger:= TRUE;
				SC_P4_Vytah.IdleTime.IN:= TRUE;
				SC_P4_Vytah.Switch1:= TRUE;
			END_IF

			IF CAM16.STAV.Results_READY AND CAM16.STAV.Command_AKCEPTOVANY AND CAM16.STAV.OldRunCounter <> CAM16.STAV.RunCounter THEN
				PocetTrigrovKamery:= 0;
				CAM16.STAV.Results_READY:= FALSE;
				CAM16.STAV.OldRunCounter:= CAM16.STAV.RunCounter;
				P4_Vytah.CMD.Banner_LED_OFF:= TRUE;
				IF NOT Linka.PAR.VyprazdnenieLinky THEN
					SC_P4_Vytah.ResetStep:= TRUE;
					SC_P4_Vytah.Step:= 135;
				ELSE
					SC_P4_Vytah.ResetStep:= TRUE;
					SC_P4_Vytah.Step:= 136;
				END_IF
			ELSIF SC_P4_Vytah.IdleTime.Q AND PocetTrigrovKamery < 5 THEN
				PocetTrigrovKamery:= PocetTrigrovKamery + 1;
				CAM16.CMD.Triger:= FALSE;
				CAM16.STAV.Results_READY:= FALSE;
				CAM16.STAV.OldRunCounter:= CAM16.STAV.RunCounter;
				P4_Vytah.CMD.Banner_LED_OFF:= TRUE;
				SC_P4_Vytah.ResetStep:= TRUE;
				SC_P4_Vytah.Step:= 134;
			ELSIF SC_P4_Vytah.IdleTime.Q AND PocetTrigrovKamery >= 5 THEN
				P34_Alarmy[455]:= TRUE;
				P4_Pracovisko.STAV.Porucha_ST6:= TRUE;
			END_IF

		134:
			SC_P4_Vytah.StepName:='134 - Automaticky Rezim - cakam na opatovny triger kamery CAM16';
			SC_P4_Vytah.IdleTime.PT:= T#2s;
			SC_P4_Vytah.AlarmTime.PT:= T#5s;

			SC_P4_Vytah.IdleTime.IN:= TRUE;

			IF SC_P4_Vytah.IdleTime.Q THEN
				SC_P4_Vytah.ResetStep:= TRUE;
				SC_P4_Vytah.Step:= 133;
			END_IF

		135:
			SC_P4_Vytah.StepName:='135 - Automaticky Rezim - kontrola vysledku kamery';
			SC_P4_Vytah.IdleTime.PT:= T#200ms;
			SC_P4_Vytah.AlarmTime.PT:= T#5s;
			SC_P4_Vytah.IdleTime.IN:= TRUE;

			IF Linka.P4_Kamery_OFF THEN
				CAM16.CMD.Triger:= FALSE;
				CAM16.PAR.ResultFotky:= 'PASS';
				SC_P4_Vytah.ResetStep:= TRUE;
				SC_P4_Vytah.Step:= 138;
			ELSIF NOT CAM16.STAV.BUSY THEN
				CAM16.CMD.Triger:= FALSE;
				IF Linka.PAR.ZvolenyModel = '4F' THEN
					IF CAM16.RESULT.Paletka.Pritomn_Busbarov_4F AND
						CAM16.RESULT.Paletka.Pritomn_LavyMVcase AND
						CAM16.RESULT.Paletka.Pritomn_PravyMVcase AND
						NOT CAM16.RESULT.Paletka.Pritomn_PowerCP THEN
						CAM16.PAR.ResultFotky:= 'PASS';
					ELSE
						CAM16.PAR.ResultFotky:= 'FAIL';
					END_IF
				ELSIF Linka.PAR.ZvolenyModel = '5F' THEN
					IF CAM16.RESULT.Paletka.Pritomn_Busbarov_5F AND
						CAM16.RESULT.Paletka.Pritomn_LavyMVcase AND
						CAM16.RESULT.Paletka.Pritomn_PravyMVcase AND
						NOT CAM16.RESULT.Paletka.Pritomn_PowerCP THEN
						CAM16.PAR.ResultFotky:= 'PASS';
					ELSE
						CAM16.PAR.ResultFotky:= 'FAIL';
					END_IF
				ELSIF Linka.PAR.ZvolenyModel = '5H' THEN
					IF CAM16.RESULT.Paletka.Pritomn_Busbarov_5H AND
						CAM16.RESULT.Paletka.Pritomn_LavyMVcase AND
						CAM16.RESULT.Paletka.Pritomn_PravyMVcase AND
						NOT CAM16.RESULT.Paletka.Pritomn_PowerCP THEN
						CAM16.PAR.ResultFotky:= 'PASS';
					ELSE
						CAM16.PAR.ResultFotky:= 'FAIL';
					END_IF
				END_IF
				SC_P4_Vytah.ResetStep:= TRUE;
				SC_P4_Vytah.Step:= 138;
			END_IF

		136:
			SC_P4_Vytah.StepName:='136 - Automaticky Rezim - kontrola vysledku kamery pri vyprazdneni linky';
			SC_P4_Vytah.IdleTime.PT:= T#200ms;
			SC_P4_Vytah.AlarmTime.PT:= T#5s;
			SC_P4_Vytah.IdleTime.IN:= TRUE;

			IF NOT CAM16.STAV.BUSY THEN
				CAM16.CMD.Triger:= FALSE;
				IF NOT CAM16.RESULT.Paletka.Pritomn_Busbarov_4F AND
					NOT CAM16.RESULT.Paletka.Pritomn_Busbarov_5F AND
					NOT CAM16.RESULT.Paletka.Pritomn_Busbarov_5H AND
					NOT	CAM16.RESULT.Paletka.Pritomn_LavyMVcase AND
					NOT	CAM16.RESULT.Paletka.Pritomn_PravyMVcase AND
					NOT CAM16.RESULT.Paletka.Pritomn_PowerCP THEN
					CAM16.PAR.ResultFotky:= 'PASS';
				ELSE
					CAM16.PAR.ResultFotky:= 'FAIL';
				END_IF
				SC_P4_Vytah.ResetStep:= TRUE;
				SC_P4_Vytah.Step:= 138;
			END_IF

		138:
			SC_P4_Vytah.StepName:='138 - Automaticky Rezim - vymazanie adresara kamery';
			SC_P4_Vytah.IdleTime.PT:= T#4s;
			SC_P4_Vytah.AlarmTime.PT:= T#5s;

			P4_Vytah.Banner.IN.ModraLED_ON:= TRUE;

			IF Linka.KOM_FTP_OFF THEN
				P4_Vytah.CMD.Banner_LED_OFF:= TRUE;
				SC_P4_Vytah.ResetStep:= TRUE;
				SC_P4_Vytah.Step:= 140;
			ELSIF NOT SC_P4_Vytah.Switch1 THEN
				FTP_CAM16.CMD.VymazFotku:= TRUE;
				SC_P4_Vytah.Switch1:= TRUE;
			END_IF

			IF FTP_CAM16.STATUS.KomunikaciaUkoncena THEN
				P4_Vytah.CMD.Banner_LED_OFF:= TRUE;
				FTP_CAM16.CMD.VymazFotku:= FALSE;
				SC_P4_Vytah.ResetStep:= TRUE;
				SC_P4_Vytah.Step:= 140;
			ELSIF FTP_CAM16.STATUS.KomunikaciaError THEN
				P34_Alarmy[410]:= TRUE;
				P4_Pracovisko.STAV.Porucha_ST6:= TRUE;
			END_IF

		140:
			SC_P4_Vytah.StepName:='140 - Automaticky Rezim - rozhodnutie podla kamerovej kontroly paletky';
			SC_P4_Vytah.IdleTime.PT:= T#200ms;
			SC_P4_Vytah.AlarmTime.PT:= T#5s;

			IF CAM16.PAR.ResultFotky = 'PASS' THEN
				SC_P4_Vytah.ResetStep:= TRUE;
				SC_P4_Vytah.Step:= 560;
			ELSIF CAM16.PAR.ResultFotky = 'FAIL' THEN
				SC_P4_Vytah.ResetStep:= TRUE;
				SC_P4_Vytah.Step:= 143;
			END_IF

		143:
			SC_P4_Vytah.StepName:='143 - Automaticky Rezim - zobrazenie hlasenia naloz spravny material na paletku';
			SC_P4_Vytah.IdleTime.PT:= T#200ms;
			SC_P4_Vytah.AlarmTime.PT:= T#5s;

			P4_Vytah.Banner.IN.CervenaLED_ON:= Blikac500ms;

			IF NOT SC_P4_Vytah.Switch1 THEN
				IF Linka.PAR.VyprazdnenieLinky THEN
					P34_Vizu.ZobrazHL4_ST10:= TRUE;
				ELSIF Linka.PAR.ZvolenyModel = '4F' THEN
					P34_Vizu.ZobrazHL1_ST10:= TRUE;
				ELSIF Linka.PAR.ZvolenyModel = '5F' THEN
					P34_Vizu.ZobrazHL2_ST10:= TRUE;
				ELSIF Linka.PAR.ZvolenyModel = '5H' THEN
					P34_Vizu.ZobrazHL3_ST10:= TRUE;
				END_IF
				SC_P4_Vytah.Switch1:= TRUE;
			END_IF

			IF P4_Vytah.Banner.OUT.Stlaceny THEN
				P34_Vizu.ZobrazHL1_ST10:= FALSE;
				P34_Vizu.ZobrazHL2_ST10:= FALSE;
				P34_Vizu.ZobrazHL3_ST10:= FALSE;
				P34_Vizu.ZobrazHL4_ST10:= FALSE;
				P4_Vytah.CMD.Banner_LED_OFF:= TRUE; //Zhasnem banner
				SC_P4_Vytah.ResetStep:= TRUE;
				SC_P4_Vytah.Step:= 130;
			ELSIF P4_Vytah_KAM_Result_Ignoruj THEN
				P4_Vytah_KAM_Result_Ignoruj:= FALSE;
				P34_Vizu.ZobrazHL1_ST10:= FALSE;
				P34_Vizu.ZobrazHL2_ST10:= FALSE;
				P34_Vizu.ZobrazHL3_ST10:= FALSE;
				P34_Vizu.ZobrazHL4_ST10:= FALSE;
				P4_Vytah.CMD.Banner_LED_OFF:= TRUE; //Zhasnem banner
				SC_P4_Vytah.ResetStep:= TRUE;
				SC_P4_Vytah.Step:= 560;
			END_IF

			//***********************************Vyvezenie paletky****************************************//
		560:
			SC_P4_Vytah.StepName:='560 - Automaticky Rezim - cakam na vyvezenie na spodny dopravnik';
			SC_P4_Vytah.IdleTime.PT:= T#1s;
			SC_P4_Vytah.AlarmTime.PT:= T#5s;

			SC_P4_Vytah.IdleTime.IN:= NOT P4_SpodnyStoper.IN.ZaplnenieDopravnika;
			P34_Vizu.ZobrazHL6_ST10:= NOT Safety.STAV.P4_Vytah_Bariera_AKTIVNA;

			IF P4_Vytah.KoniecCyklu THEN
				SC_P4_Vytah.ResetStep:= TRUE;
				SC_P4_Vytah.Step:= 0;
			ELSIF SC_P4_Vytah.IdleTime.Q AND P4_Vytah.RFID_hlava.PritomnostPaletky AND Safety.STAV.P4_Vytah_Bariera_AKTIVNA AND NOT P4_Vytah.IN.PrechodDopravnika THEN
				Paletka[i].PAR.CisloPaletky:= '';
				Paletka[i].STAV.StavPaletky:= '';
				Paletka[i].STAV.TypModelu:= '';
				Paletka[i].STAV.KodModelu:= '';
				Paletka[i].PAR.QRkodFiltra_4F5F:= '';
				Paletka[i].PAR.QRkodFiltra_5H:= '';
				Paletka[i].PAR.QRkodPowerCP:= '';
				Paletka[i].PAR.StavPowerCP:= '';
				Paletka[i].STAV.CisloTestovacejStanice:= '';
				Paletka[i].STAV.CisloRevorkovejStanice:= '';
				Paletka[i].PAR.ID_Operatora:= '';
				Paletka[i].STAV.Komunikacia_DONE:= FALSE;
				Paletka[i].STAV.OdoslanieFotiek_DONE:= FALSE;
				Paletka[i].STAV.CisloEtiketyVyziadane:= FALSE;
				Paletka[i].STAV.FunkcnyTest_Ukonceny:= FALSE;
				Paletka[i].STAV.HV_Test_Ukonceny:= FALSE;
				Paletka[i].STAV.LeakageTest_Ukonceny:= FALSE;
				Paletka[i].STAV.QRkodFiltraPriradeny:= FALSE;
				Paletka[i].STAV.Zvaranie_Ukoncene:= FALSE;
				Paletka[i].STAV.NalepenieEtikety_DONE:= FALSE;
				CisloFotky:= 0;
				Reports.Kamery.P4_CAM16_KontrolaPaletky:= '';
				P4_Vytah.CMD.Banner_LED_OFF:= TRUE;
				P34_Vizu.ZobrazHL6_ST10:= FALSE;
				SC_P4_Vytah.ResetStep:= TRUE;
				SC_P4_Vytah.Step:= 563;
			ELSIF NOT P4_Vytah.RFID_hlava.PritomnostPaletky THEN
				P34_Vizu.ZobrazHL6_ST10:= FALSE;
				SC_P4_Vytah.ResetStep:= TRUE;
				SC_P4_Vytah.Step:= 100;
			END_IF

		563:
			SC_P4_Vytah.StepName:='563 - Automaticky Rezim - presuvam vytah do spodnej pozicie vyvazania';
			SC_P4_Vytah.IdleTime.PT:= T#1s;
			SC_P4_Vytah.AlarmTime.PT:= T#5s;

			SC_P4_Vytah.IdleTime.IN:= Safety.STAV.P4_Vytah_Bariera_AKTIVNA;
			P34_Vizu.ZobrazHL6_ST10:= NOT Safety.STAV.P4_Vytah_Bariera_AKTIVNA;

			P4_Vytah.ServoZdvihuVytahu.Parameters.Velocity:= P34_RemPremenne.P4_Vytah_RychlostZdvihu/1000;
			P4_Vytah.ServoZdvihuVytahu.Parameters.Position:= P34_RemPremenne.P4_Vytah_PoziciaVykladania;
			ServoZdvihu_ZadanaPozicia_UDINT:= REAL_TO_UDINT(P34_RemPremenne.P4_Vytah_PoziciaVykladania);

			P4_Vytah.Banner.IN.OranzovaLED_ON:= Blikac1s;

			IF NOT SC_P4_Vytah.Switch1 AND SC_P4_Vytah.IdleTime.Q THEN
				P4_Vytah.ServoZdvihuVytahu.Command.MovePosition:= TRUE;
				P34_Vizu.ZobrazHL6_ST10:= FALSE;
				SC_P4_Vytah.Switch1:= TRUE;
			END_IF

			IF P4_Vytah.ServoZdvihuVytahu.Status.InPosition AND (ServoZdvihu_AktualPosition_UDINT = ServoZdvihu_ZadanaPozicia_UDINT) THEN
				P4_Vytah.ServoZdvihuVytahu.Command.MovePosition:= FALSE;
				SC_P4_Vytah.ResetStep:= TRUE;
				SC_P4_Vytah.Step:= 565;
			END_IF

		565:
			SC_P4_Vytah.StepName:='565 - Automaticky Rezim - vyvazam na spodny dopravnik';
			SC_P4_Vytah.IdleTime.PT:= T#3s;
			SC_P4_Vytah.AlarmTime.PT:= T#5s;

			P4_Vytah.Banner.IN.OranzovaLED_ON:= Blikac1s;

			IF P4_Dopravniky.STAV.PoINIT THEN
				P4_Vytah.OUT.DopravnikChod_VZAD:= TRUE;
				SC_P4_Vytah.ResetStep:= TRUE;
				SC_P4_Vytah.Step:= 568;
			END_IF

		568:
			SC_P4_Vytah.StepName:='568 - Automaticky Rezim - ukoncenie vyvazania na spodny dopravnik';
			SC_P4_Vytah.IdleTime.PT:= T#400ms;
			SC_P4_Vytah.AlarmTime.PT:= T#5s;

			P4_Vytah.Banner.IN.OranzovaLED_ON:= Blikac1s;

			IF EDGEPOS(P4_Vytah.IN.PrechodDopravnika) THEN
				SC_P4_Vytah.IdleTime.IN:= TRUE;
			END_IF

			IF SC_P4_Vytah.IdleTime.Q AND NOT P4_Vytah.IN.PrechodDopravnika AND NOT P4_Vytah.RFID_hlava.PritomnostPaletky THEN
				P4_Vytah.OUT.DopravnikChod_VZAD:= FALSE;
				SC_P4_Vytah.ResetStep:= TRUE;
				SC_P4_Vytah.Step:= 570;
			END_IF

		570:
			SC_P4_Vytah.StepName:='570 - Automaticky Rezim - cakam na spustenie presunu vytahu do hornej pozicie navazania';
			SC_P4_Vytah.IdleTime.PT:= T#100ms;
			SC_P4_Vytah.AlarmTime.PT:= T#5s;

			P4_Vytah.Banner.IN.OranzovaLED_ON:= Blikac1s;

			SC_P4_Vytah.IdleTime.IN:= Safety.STAV.P4_Vytah_Bariera_AKTIVNA AND NOT P4_Vytah.IN.PrechodDopravnika AND NOT P4_Vytah.RFID_hlava.PritomnostPaletky;
			P34_Vizu.ZobrazHL6_ST10:= NOT Safety.STAV.P4_Vytah_Bariera_AKTIVNA;

			IF SC_P4_Vytah.IdleTime.Q  THEN
				P34_Vizu.ZobrazHL6_ST10:= FALSE;
				SC_P4_Vytah.ResetStep:= TRUE;
				SC_P4_Vytah.Step:= 573;
			END_IF

		573:
			SC_P4_Vytah.StepName:='573 - Automaticky Rezim - presuvam vytah do hornej pozicie navazania';
			SC_P4_Vytah.IdleTime.PT:= T#200ms;
			SC_P4_Vytah.AlarmTime.PT:= T#5s;

			P4_Vytah.Banner.IN.OranzovaLED_ON:= Blikac1s;

			P4_Vytah.ServoZdvihuVytahu.Parameters.Velocity:= P34_RemPremenne.P4_Vytah_RychlostZdvihu/1000;
			P4_Vytah.ServoZdvihuVytahu.Parameters.Position:= P34_RemPremenne.P4_Vytah_PoziciaNakladania;

			IF NOT SC_P4_Vytah.Switch1 THEN
				P4_Vytah.ServoZdvihuVytahu.Command.MovePosition:= TRUE;
				SC_P4_Vytah.Switch1:= TRUE;
			END_IF

			IF EDGEPOS(P4_Vytah.ServoZdvihuVytahu.Status.InPosition) THEN
				P4_Vytah.ServoZdvihuVytahu.Command.MovePosition:= FALSE;
				P4_Vytah.CMD.Banner_LED_OFF:= TRUE;
				SC_P4_Vytah.ResetStep:= TRUE;
				SC_P4_Vytah.Step:= 100;
			END_IF

			//*******************************************************Manuálny režim*******************************************************************************//
		700:
			SC_P4_Vytah.StepName:='700 - Manualny Rezim';
			SC_P4_Vytah.IdleTime.PT:= T#8s;
			SC_P4_Vytah.AlarmTime.PT:= T#5s;

			//Ovládanie zdvihu výťahu//
			P4_Vytah.ServoZdvihuVytahu.Parameters.Acc:= 10;
			P4_Vytah.ServoZdvihuVytahu.Parameters.Dcc:= 50;
			P4_Vytah.ServoZdvihuVytahu.Parameters.Velocity:= P4_Vytah.PAR.Zdvih_JoggRychlost/1000;
			P4_Vytah.ServoZdvihuVytahu.Command.TorqueLimitation:= TRUE;
			P4_Vytah.ServoZdvihuVytahu.Parameters.Torque:= 1.5;

			IF P4_Vytah.CMD.RR_ZdvihVytahu_DOLE AND NOT P4_Vytah.ServoZdvihuVytahu.Command.Stop THEN
				P4_Vytah.ServoZdvihuVytahu.Parameters.Position:= P34_RemPremenne.P4_Vytah_PoziciaVykladania;
				P4_Vytah.ServoZdvihuVytahu.Command.MovePosition:= TRUE;
			ELSIF P4_Vytah.CMD.RR_ZdvihVytahu_HORE AND NOT P4_Vytah.ServoZdvihuVytahu.Command.Stop THEN
				P4_Vytah.ServoZdvihuVytahu.Parameters.Position:= P34_RemPremenne.P4_Vytah_PoziciaNakladania;
				P4_Vytah.ServoZdvihuVytahu.Command.MovePosition:= TRUE;
			ELSE
				P4_Vytah.ServoZdvihuVytahu.Command.MovePosition:= FALSE;
				P4_Vytah.ServoZdvihuVytahu.Command.Stop:= TRUE;
			END_IF

			IF P4_Vytah.ServoZdvihuVytahu.Command.Stop AND P4_Vytah.ServoZdvihuVytahu.Status.StandStill THEN
				P4_Vytah.ServoZdvihuVytahu.Command.Stop:= FALSE;
			END_IF

			//Ovládanie dopravníka výťahu//
			IF P4_Vytah.CMD.RR_ChodDopravnika_VPRED THEN
				P4_Vytah.OUT.DopravnikChod_VZAD:= FALSE;
				P4_Vytah.OUT.DopravnikChod_VPRED:= TRUE;
			ELSIF P4_Vytah.CMD.RR_ChodDopravnika_VZAD THEN
				P4_Vytah.OUT.DopravnikChod_VPRED:= FALSE;
				P4_Vytah.OUT.DopravnikChod_VZAD:= TRUE;
			ELSE
				P4_Vytah.OUT.DopravnikChod_VPRED:= FALSE;
				P4_Vytah.OUT.DopravnikChod_VZAD:= FALSE;
			END_IF

			//Čítanie a zápis na paletku//
			IF P4_Vytah.RFID_hlava.PrecitajChipRFID AND (P4_Vytah.RFID_hlava.Stav_CitanieZapis_OK OR P4_Vytah.RFID_hlava.Stav_CitanieZapis_NG) THEN
				P4_Vytah.PAR.RR_PrecitaneCisloPaletky:= P4_Vytah.RFID_hlava.PrecitaneCisloPaletky;
				P4_Vytah.RFID_hlava.PrecitajChipRFID:= FALSE;
			END_IF

			IF P4_Vytah.RFID_hlava.ZapisNaChipRFID AND (P4_Vytah.RFID_hlava.Stav_CitanieZapis_OK OR P4_Vytah.RFID_hlava.Stav_CitanieZapis_NG) THEN
				P4_Vytah.RFID_hlava.ZapisNaChipRFID:= FALSE;
			END_IF

	END_CASE

				END_PROGRAM

PROGRAM _EXIT
				(* Insert code here *)

				END_PROGRAM
```

#### Variables.var - Local variables
```iecst
VAR
	PocetTrigrovKamery : USINT := 0;
	PocetDopytovNaServer : USINT := 0;
	CisloFotky : USINT := 0;
	TestovaciKus : BOOL := 0;
	i : USINT := 0;
	Stav_VlozenaPaletka : BOOL := 0;
	CasEnable_1 : TON;
	CasResetServo_1 : TON;
	ServoZdvihu_AktualPosition_UDINT : UDINT := 0;
	ServoZdvihu_ZadanaPozicia_UDINT : UDINT := 0;
END_VAR
```

#### IOLinkKomunikacia.st
```iecst
ACTION IOLinkKomunikacia:

	//RFID snímač paletky//
	P4_Vytah.RFID_hlava();

	//Ovládanie bannera//
	P4_Vytah.Banner.IN.Blikac100ms:= Blikac500ms;
	P4_Vytah.Banner();

END_ACTION
```

### Program Logical/Program/Pracovisko_4/P4_OvladVizu (IEC)

#### Main.st - Init, cyclic, exit code
```iecst
PROGRAM _INIT
	(* Insert code here *)

END_PROGRAM

PROGRAM _CYCLIC

	//*************************************Prepnutie obrazovky pri stlačení tlačítka CS*********************************//
	IF EDGEPOS(P3_Pracovisko.STAV.Manual AND NOT Safety.STAV.Linka_ZonaCS_AKTIVNA) THEN
		P34_Vizu.GoPage:= 'PageAutomatP34';
	ELSIF EDGEPOS(P4_Pracovisko.STAV.Manual AND NOT Safety.STAV.Linka_ZonaCS_AKTIVNA) THEN
		P34_Vizu.GoPage:= 'PageAutomatP34';
	END_IF

	//************************************Filter alarmov**************************************************************//
	FilterVizu_P34:= '[{"logicalOperator":"and","value":300,"conditionType":">=","columnType":"cod","useAlarmState":false,"alarmState":0},{"value":500,"conditionType":"<=","columnType":"cod","useAlarmState":false,"alarmState":0}]';

	//***********************Prepnutie bootovacej obrazovky********************************//
	IF P34_Vizu.ActualPage <> 'PageBootP34' AND NOT Safety.STAV.Linka_SafetyPLC_Nabehlo THEN
		P34_Vizu.GoPage:= 'PageBootP34';
	ELSIF P34_Vizu.ActualPage = 'PageBootP34' AND Safety.STAV.Linka_SafetyPLC_Nabehlo THEN
		P34_Vizu.GoPage:= 'PageAutomatP34';
	END_IF

	IF P34_Vizu.GoPage = 'PageBootP34' AND P34_Vizu.ActualPage = 'PageBootP34' THEN
		P34_Vizu.GoPage:= '';
	ELSIF P34_Vizu.GoPage = 'PageAutomatP34' AND P34_Vizu.ActualPage = 'PageAutomatP34' THEN
		P34_Vizu.GoPage:= '';
	END_IF

	//********************************Blikanie tlačítka Alarmy*******************************************************//
	IF (P3_Pracovisko.STAV.PORUCHA OR P4_Pracovisko.STAV.PORUCHA) AND P34_Vizu.ActualPage <> 'PageAlarmP34' THEN
		IF Blikac500ms THEN
			P34_AlarmyVizu.FarbaTlacitka_Alarmy:= "Button_Red";
		ELSE
			P34_AlarmyVizu.FarbaTlacitka_Alarmy:= "default";
		END_IF
	ELSE
		P34_AlarmyVizu.FarbaTlacitka_Alarmy:= "default";
	END_IF

	//*****************************************BUNKA 3*********************************************************//

	//********Zmeny farieb tlačítok ovládania zámkov bunky 3***************//
	//Zadné dvere //
	IF P3_Pracovisko.STAV.ZadneDvereZamknute AND P3_Pracovisko.IN.ZadneDvereLave_PritomnAdaptera AND P3_Pracovisko.IN.ZadneDverePrave_PritomnAdaptera THEN
		P34_Vizu.TL_ZadnyZamok_Farba_P3:= "Button_Green";
	ELSIF P3_Pracovisko.IN.ZadneDvereLave_PritomnAdaptera AND P3_Pracovisko.IN.ZadneDverePrave_PritomnAdaptera THEN
		IF Blikac1s THEN
			P34_Vizu.TL_ZadnyZamok_Farba_P3:= "Button_Blue";
		ELSE
			P34_Vizu.TL_ZadnyZamok_Farba_P3:= "Operate";
		END_IF
	ELSE
		P34_Vizu.TL_ZadnyZamok_Farba_P3:= "Button_Red";
	END_IF

	//Predné dvere //
	IF P3_Pracovisko.STAV.PredneDvereZamknute AND P3_Pracovisko.IN.PredneDvereLave_PritomnAdaptera AND P3_Pracovisko.IN.PredneDverePrave_PritomnAdaptera THEN
		P34_Vizu.TL_PrednyZamok_Farba_P3:= "Button_Green";
	ELSIF P3_Pracovisko.IN.PredneDvereLave_PritomnAdaptera AND P3_Pracovisko.IN.PredneDverePrave_PritomnAdaptera THEN
		IF Blikac1s THEN
			P34_Vizu.TL_PrednyZamok_Farba_P3:= "Button_Blue";
		ELSE
			P34_Vizu.TL_PrednyZamok_Farba_P3:= "Operate";
		END_IF
	ELSE
		P34_Vizu.TL_PrednyZamok_Farba_P3:= "Button_Red";
	END_IF

	//************Zobrazenie warningov bunky 3**********************//
	//0 - Pracovisko je vypnuté.
	//1 - Prebieha inicializácia pracoviska.
	//2 - Na pracovisku prebieha výroba.
	//3 - Prebieha ukončenie pracovného cyklu pracoviska.
	//4 - Prebieha režim vyprázdnenia linky.
	//5 - Doplň zásobník skrutiek K40 !!!
	//6 - Doplň zásobník skrutiek M5 !!!
	//7 - Niesu založené správne kontakty na HV teste !!!
	//8 - Niesu založené správne kontakty na Leakage teste stanica A !!!
	//9 - Niesu založené správne kontakty na Leakage teste stanica B !!!

	IF Linka.PAR.ZvolenyModel = '4F' AND NOT P3_HV_Test.IN.TypKonektoru_4F THEN
		P34_Vizu.WarningsP3_Index:= 7;
	ELSIF Linka.PAR.ZvolenyModel = '5F' AND NOT P3_HV_Test.IN.TypKonektoru_5F_5H THEN
		P34_Vizu.WarningsP3_Index:= 7;
	ELSIF Linka.PAR.ZvolenyModel = '5H' AND NOT P3_HV_Test.IN.TypKonektoru_5F_5H THEN
		P34_Vizu.WarningsP3_Index:= 7;
	ELSIF Linka.PAR.ZvolenyModel = '4F' AND NOT P3_LeakageTestA.IN.Tester_TypKonektoru_4F THEN
		P34_Vizu.WarningsP3_Index:= 8;
	ELSIF Linka.PAR.ZvolenyModel = '5F' AND NOT P3_LeakageTestA.IN.Tester_TypKonektoru_5F_5H THEN
		P34_Vizu.WarningsP3_Index:= 8;
	ELSIF Linka.PAR.ZvolenyModel = '5H' AND NOT P3_LeakageTestA.IN.Tester_TypKonektoru_5F_5H THEN
		P34_Vizu.WarningsP3_Index:= 8;
	ELSIF Linka.PAR.ZvolenyModel = '4F' AND NOT P3_LeakageTestB.IN.Tester_TypKonektoru_4F THEN
		P34_Vizu.WarningsP3_Index:= 9;
	ELSIF Linka.PAR.ZvolenyModel = '5F' AND NOT P3_LeakageTestB.IN.Tester_TypKonektoru_5F_5H THEN
		P34_Vizu.WarningsP3_Index:= 9;
	ELSIF Linka.PAR.ZvolenyModel = '5H' AND NOT P3_LeakageTestB.IN.Tester_TypKonektoru_5F_5H THEN
		P34_Vizu.WarningsP3_Index:= 9;
	ELSIF P3_Pracovisko.STAV.Automat AND NOT P3_Pracovisko.STAV.PoINIT AND NOT P3_Pracovisko.STAV.UkoncenieCyklu_BUSY THEN
		P34_Vizu.WarningsP3_Index:= 1;
	ELSIF P3_Srobovanie.SkrutSet_K40.IN.VibracnyHrniec.PritomnostSkrutiekVHrnci THEN
		P34_Vizu.WarningsP3_Index:= 5;
	ELSIF P3_Srobovanie.SkrutSet_M5.IN.ZasobnikSkrutiekPrazdny THEN
		P34_Vizu.WarningsP3_Index:= 6;
	ELSIF Linka.PAR.TestovaciKus THEN
		P34_Vizu.WarningsP3_Index:= 11;
	ELSIF Linka.PAR.VyprazdnenieLinky THEN
		P34_Vizu.WarningsP3_Index:= 4;
	ELSIF P3_Pracovisko.STAV.PoINIT AND NOT P3_Pracovisko.STAV.UkoncenieCyklu_BUSY THEN
		P34_Vizu.WarningsP3_Index:= 2;
	ELSIF P3_Pracovisko.STAV.UkoncenieCyklu_BUSY THEN
		P34_Vizu.WarningsP3_Index:= 3;
	ELSIF NOT P3_Pracovisko.STAV.Automat THEN
		P34_Vizu.WarningsP3_Index:= 0;
	END_IF

	//*************Prepínanie farby textového pola warning bunky 3*****************//
	IF P34_Vizu.WarningsP3_Index = 0 THEN
		P34_Vizu.WarningsP3_Farba:= "TextOutput_Grey";
	ELSIF P34_Vizu.WarningsP3_Index = 1 THEN
		P34_Vizu.WarningsP3_Farba:= "TextOutput_Blue";
	ELSIF P34_Vizu.WarningsP3_Index = 2 THEN
		P34_Vizu.WarningsP3_Farba:= "TextOutput_Green";
	ELSIF P34_Vizu.WarningsP3_Index = 3 THEN
		P34_Vizu.WarningsP3_Farba:= "TextOutput_Blue";
	ELSIF P34_Vizu.WarningsP3_Index = 4 THEN
		P34_Vizu.WarningsP3_Farba:= "TextOutput_Green";
	ELSIF P34_Vizu.WarningsP3_Index = 11 THEN
		P34_Vizu.WarningsP3_Farba:= "TextOutput_Green";
	ELSE
		IF Blikac1s THEN
			P34_Vizu.WarningsP3_Farba:= "TextOutput_Orange";
		ELSE
			P34_Vizu.WarningsP3_Farba:= "TextOutput_Grey";
		END_IF
	END_IF

	//*************Zamknutie tlačítok bunky 3************************//
	//Zamknutie tlačítok ovládania zámkov//
	IF P3_Pracovisko.STAV.Automat THEN
		P34_Vizu.TL_OvladaniaZamkov_ENABLE_P3:= FALSE;
	ELSIF P3_Srobovanie.STAV.RR_Polohovanie_BUSY THEN
		P34_Vizu.TL_OvladaniaZamkov_ENABLE_P3:= FALSE;
	ELSIF P3_Srobovanie.STAV.CistenieSkrutkovackyK40_BUSY THEN
		P34_Vizu.TL_OvladaniaZamkov_ENABLE_P3:= FALSE;
	ELSIF P3_HV_Test.STAV.RR_SekvenciaTestera_BUSY THEN
		P34_Vizu.TL_OvladaniaZamkov_ENABLE_P3:= FALSE;
	ELSIF P3_LeakageTestA.STAV.RR_TestovaciaSekvencia_BUSY THEN
		P34_Vizu.TL_OvladaniaZamkov_ENABLE_P3:= FALSE;
	ELSIF P3_LeakageTestB.STAV.RR_TestovaciaSekvencia_BUSY THEN
		P34_Vizu.TL_OvladaniaZamkov_ENABLE_P3:= FALSE;
	ELSE
		P34_Vizu.TL_OvladaniaZamkov_ENABLE_P3:= TRUE;
	END_IF

	//Tlačítko Štat Automat//
	IF P3_Pracovisko.STAV.UkoncenieCyklu_BUSY THEN
		P34_Vizu.TL_StartAutomat_ENABLE_P3:= FALSE;
	ELSIF P3_Pracovisko.STAV.PORUCHA THEN
		P34_Vizu.TL_StartAutomat_ENABLE_P3:= FALSE;
	ELSIF NOT Safety.STAV.P3_ZonaBunky_AKTIVNA THEN
		P34_Vizu.TL_StartAutomat_ENABLE_P3:= FALSE;
	ELSIF NOT P3_Pracovisko.STAV.HardwareBunky_OK THEN
		P34_Vizu.TL_StartAutomat_ENABLE_P3:= FALSE;
	ELSE
		P34_Vizu.TL_StartAutomat_ENABLE_P3:= TRUE;
	END_IF

	//Tlačítko Ukončenie Cyklu//
	IF P3_Pracovisko.STAV.PoINIT THEN
		P34_Vizu.TL_KoniecCyklu_ENABLE_P3:= TRUE;
	ELSE
		P34_Vizu.TL_KoniecCyklu_ENABLE_P3:= FALSE;
	END_IF

	//Tlačítko STOP//
	IF P3_Pracovisko.STAV.PoINIT AND NOT P3_Pracovisko.STAV.UkoncenieCyklu_BUSY THEN
		P34_Vizu.TL_STOP_ENABLE_P3:= FALSE;
	ELSE
		P34_Vizu.TL_STOP_ENABLE_P3:= TRUE;
	END_IF

	//Tlačítko Režim Manual//
	IF P3_Pracovisko.STAV.Automat THEN
		P34_Vizu.TL_RezimManual_ENABLE_P3:= FALSE;
	ELSIF NOT P3_Pracovisko.STAV.HardwareBunky_OK THEN
		P34_Vizu.TL_RezimManual_ENABLE_P3:= FALSE;
	ELSE
		P34_Vizu.TL_RezimManual_ENABLE_P3:= TRUE;
	END_IF

	//Tlačítka vypnutia leakage testov//
//	IF P3_Pracovisko.STAV.Automat THEN
//		P34_Vizu.VolbaLeakageTestu_ENABLE:= FALSE;
//	ELSE
		P34_Vizu.VolbaLeakageTestu_ENABLE:= TRUE;
//	END_IF

	//RR - Tlačítko čistenia skrutkovačky K40//
	IF P3_Srobovanie.STAV.RR_Polohovanie_BUSY THEN
		P34_Vizu.TL_VycistiSkrutkovackuK40_ENABLE:= FALSE;
	ELSIF NOT Safety.STAV.P3_ZonaBunky_AKTIVNA THEN
		P34_Vizu.TL_VycistiSkrutkovackuK40_ENABLE:= FALSE;
	ELSIF NOT Safety.STAV.Linka_ZonaCS_AKTIVNA THEN
		P34_Vizu.TL_VycistiSkrutkovackuK40_ENABLE:= FALSE;
	ELSIF P3_Srobovanie.STAV.CistenieSkrutkovackyK40_BUSY THEN
		P34_Vizu.TL_VycistiSkrutkovackuK40_ENABLE:= FALSE;
	ELSIF NOT P3_Pracovisko.STAV.SkrutkovackyZasunute THEN
		P34_Vizu.TL_VycistiSkrutkovackuK40_ENABLE:= FALSE;
	ELSIF P3_Srobovanie.CMD.RR_SkrutSetK40_VysunBrzdu THEN
		P34_Vizu.TL_VycistiSkrutkovackuK40_ENABLE:= FALSE;
	ELSIF P3_Srobovanie.CMD.RR_SkrutSetK40_Zasobnik_RUN THEN
		P34_Vizu.TL_VycistiSkrutkovackuK40_ENABLE:= FALSE;
	ELSE
		P34_Vizu.TL_VycistiSkrutkovackuK40_ENABLE:= TRUE;
	END_IF

	//RR - Tlačítko polohovania aplikátora//
	IF P3_Srobovanie.STAV.RR_Polohovanie_BUSY THEN
		P34_Vizu.TL_PolohujManipulator_ENABLE:= FALSE;
	ELSIF NOT Safety.STAV.P3_ZonaBunky_AKTIVNA THEN
		P34_Vizu.TL_PolohujManipulator_ENABLE:= FALSE;
	ELSIF NOT Safety.STAV.Linka_ZonaCS_AKTIVNA THEN
		P34_Vizu.TL_PolohujManipulator_ENABLE:= FALSE;
	ELSIF P3_Srobovanie.STAV.CistenieSkrutkovackyK40_BUSY THEN
		P34_Vizu.TL_PolohujManipulator_ENABLE:= FALSE;
	ELSIF NOT P3_Pracovisko.STAV.SkrutkovackyZasunute THEN
		P34_Vizu.TL_PolohujManipulator_ENABLE:= FALSE;
	ELSE
		P34_Vizu.TL_PolohujManipulator_ENABLE:= TRUE;
	END_IF

	//RR - Tlačítko vysunutia skrutkovačky K40//
	IF P3_Srobovanie.STAV.RR_Polohovanie_BUSY THEN
		P34_Vizu.Tl_VysunutieSkrutkovK40_ENABLE:= FALSE;
	ELSIF P3_Srobovanie.STAV.CistenieSkrutkovackyK40_BUSY THEN
		P34_Vizu.Tl_VysunutieSkrutkovK40_ENABLE:= FALSE;
	ELSIF NOT Safety.STAV.P3_ZonaBunky_AKTIVNA THEN
		P34_Vizu.Tl_VysunutieSkrutkovK40_ENABLE:= FALSE;
	ELSIF NOT Safety.STAV.Linka_ZonaCS_AKTIVNA THEN
		P34_Vizu.Tl_VysunutieSkrutkovK40_ENABLE:= FALSE;
	ELSE
		P34_Vizu.Tl_VysunutieSkrutkovK40_ENABLE:= TRUE;
	END_IF

	//RR - Tlačítko vysunutia skrutkovačky M5//
	IF P3_Srobovanie.STAV.RR_Polohovanie_BUSY THEN
		P34_Vizu.TL_OvladaniaVysunSkrutkovM5:= FALSE;
	ELSIF P3_Srobovanie.STAV.CistenieSkrutkovackyK40_BUSY THEN
		P34_Vizu.TL_OvladaniaVysunSkrutkovM5:= FALSE;
	ELSIF NOT Safety.STAV.P3_ZonaBunky_AKTIVNA THEN
		P34_Vizu.TL_OvladaniaVysunSkrutkovM5:= FALSE;
	ELSIF NOT Safety.STAV.Linka_ZonaCS_AKTIVNA THEN
		P34_Vizu.TL_OvladaniaVysunSkrutkovM5:= FALSE;
	ELSE
		P34_Vizu.TL_OvladaniaVysunSkrutkovM5:= TRUE;
	END_IF

	//RR - Ovládanie skrutkovacieho setu K40//
	IF P3_Srobovanie.STAV.CistenieSkrutkovackyK40_BUSY THEN
		P34_Vizu.TL_OvladSkrutkovSetuK40_ENABLE:= FALSE;
	ELSE
		P34_Vizu.TL_OvladSkrutkovSetuK40_ENABLE:= TRUE;
	END_IF

	//RR - Ovládanie manipulatora Y//
	IF NOT Safety.STAV.P3_ZonaBunky_AKTIVNA THEN
		P34_Vizu.TL_OvladManipulatoraY_ENABLE:= FALSE;
	ELSE
		P34_Vizu.TL_OvladManipulatoraY_ENABLE:= TRUE;
	END_IF

	//RR - Ovládanie HV Testu//
	IF P3_HV_Test.STAV.RR_SekvenciaTestera_BUSY THEN
		P34_Vizu.TL_OvladaniaHV_Testu_ENABLE:= FALSE;
	ELSIF NOT Safety.STAV.P3_ZonaBunky_AKTIVNA THEN
		P34_Vizu.TL_OvladaniaHV_Testu_ENABLE:= FALSE;
	ELSIF NOT Safety.STAV.Linka_ZonaCS_AKTIVNA THEN
		P34_Vizu.TL_OvladaniaHV_Testu_ENABLE:= FALSE;
	ELSE
		P34_Vizu.TL_OvladaniaHV_Testu_ENABLE:= TRUE;
	END_IF

	//RR - Ovládanie sekvencie HV Testu//
	IF NOT Safety.STAV.P3_ZonaBunky_AKTIVNA THEN
		P34_Vizu.TL_SekvencieHV_Testu_ENABLE:= FALSE;
	ELSIF NOT Safety.STAV.Linka_ZonaCS_AKTIVNA THEN
		P34_Vizu.TL_SekvencieHV_Testu_ENABLE:= FALSE;
	ELSIF NOT P3_HV_Test.RFID_hlava.PritomnostPaletky THEN
		P34_Vizu.TL_SekvencieHV_Testu_ENABLE:= FALSE;
	ELSE
		P34_Vizu.TL_SekvencieHV_Testu_ENABLE:= TRUE;
	END_IF

	//RR - Ovládanie Leakage Testu A//
	IF P3_LeakageTestA.STAV.RR_TestovaciaSekvencia_BUSY THEN
		P34_Vizu.TL_OvladaniaLeakTestuA_ENABLE:= FALSE;
	ELSIF NOT Safety.STAV.P3_ZonaBunky_AKTIVNA THEN
		P34_Vizu.TL_OvladaniaLeakTestuA_ENABLE:= FALSE;
	ELSIF NOT Safety.STAV.Linka_ZonaCS_AKTIVNA THEN
		P34_Vizu.TL_OvladaniaLeakTestuA_ENABLE:= FALSE;
	ELSE
		P34_Vizu.TL_OvladaniaLeakTestuA_ENABLE:= TRUE;
	END_IF

	//RR - Testovacia sekvencia Leakage Testu A//
	IF NOT P3_LeakageTestA.IN.HornyPritlak_ZASUNUTY OR NOT P3_LeakageTestA.IN.Centrovanie_ZASUNUTE THEN
		P34_Vizu.TL_SekvencieLeakTestuA_ENABLE:= FALSE;
	ELSIF NOT Safety.STAV.P3_ZonaBunky_AKTIVNA THEN
		P34_Vizu.TL_SekvencieLeakTestuA_ENABLE:= FALSE;
	ELSIF NOT Safety.STAV.Linka_ZonaCS_AKTIVNA THEN
		P34_Vizu.TL_SekvencieLeakTestuA_ENABLE:= FALSE;
	ELSIF P3_LeakageTestA.STAV.RR_TestovaciaSekvencia_BUSY THEN
		P34_Vizu.TL_SekvencieLeakTestuA_ENABLE:= FALSE;
	ELSIF NOT P3_LeakageTestA.RFID_hlava.PritomnostPaletky THEN
		P34_Vizu.TL_SekvencieLeakTestuA_ENABLE:= FALSE;
	ELSE
		P34_Vizu.TL_SekvencieLeakTestuA_ENABLE:= TRUE;
	END_IF

	//RR - Ovládanie Leakage Testu B//
	IF P3_LeakageTestB.STAV.RR_TestovaciaSekvencia_BUSY THEN
		P34_Vizu.TL_OvladaniaLeakTestuB_ENABLE:= FALSE;
	ELSIF NOT Safety.STAV.P3_ZonaBunky_AKTIVNA THEN
		P34_Vizu.TL_OvladaniaLeakTestuB_ENABLE:= FALSE;
	ELSIF NOT Safety.STAV.Linka_ZonaCS_AKTIVNA THEN
		P34_Vizu.TL_OvladaniaLeakTestuB_ENABLE:= FALSE;
	ELSE
		P34_Vizu.TL_OvladaniaLeakTestuB_ENABLE:= TRUE;
	END_IF

	//RR - Testovacia sekvencia Leakage Testu B//
	IF NOT P3_LeakageTestB.IN.HornyPritlak_ZASUNUTY OR NOT P3_LeakageTestB.IN.Centrovanie_ZASUNUTE THEN
		P34_Vizu.TL_SekvencieLeakTestuB_ENABLE:= FALSE;
	ELSIF NOT Safety.STAV.P3_ZonaBunky_AKTIVNA THEN
		P34_Vizu.TL_SekvencieLeakTestuB_ENABLE:= FALSE;
	ELSIF NOT Safety.STAV.Linka_ZonaCS_AKTIVNA THEN
		P34_Vizu.TL_SekvencieLeakTestuB_ENABLE:= FALSE;
	ELSIF P3_LeakageTestB.STAV.RR_TestovaciaSekvencia_BUSY THEN
		P34_Vizu.TL_SekvencieLeakTestuB_ENABLE:= FALSE;
	ELSIF NOT P3_LeakageTestB.RFID_hlava.PritomnostPaletky THEN
		P34_Vizu.TL_SekvencieLeakTestuB_ENABLE:= FALSE;
	ELSE
		P34_Vizu.TL_SekvencieLeakTestuB_ENABLE:= TRUE;
	END_IF

	//**************************Zamknutie editácie parametrov*********************************//
	IF P34_UrovenPrihlasenehoUzivatela >= 20 THEN
		P34_Vizu.EditaciaParametrov_ENABLE:= TRUE;
	ELSE
		P34_Vizu.EditaciaParametrov_ENABLE:= FALSE;
	END_IF

	//************************Prepínanie stavov pracovísk - Bunka 3***************************//
	//Dopravníky//
	IF P3_Dopravniky.Automat AND NOT P3_Dopravniky.STAV.PoINIT THEN
		P34_Vizu.IndexStavu_DopravnikP3:= 1;
	ELSIF P3_Dopravniky.Automat AND P3_Dopravniky.STAV.PoINIT THEN
		P34_Vizu.IndexStavu_DopravnikP3:= 2;
	ELSE
		P34_Vizu.IndexStavu_DopravnikP3:= 0;
	END_IF

	//Spodný stoper//
	IF P3_SpodnyStoper.Automat AND NOT P3_SpodnyStoper.STAV.PoINIT THEN
		P34_Vizu.IndexStavu_SpodnyStoperP3:= 1;
	ELSIF P3_SpodnyStoper.Automat AND P3_SpodnyStoper.STAV.PoINIT THEN
		P34_Vizu.IndexStavu_SpodnyStoperP3:= 2;
	ELSE
		P34_Vizu.IndexStavu_SpodnyStoperP3:= 0;
	END_IF

	//Stoper šrobovania//
	IF NOT P3_Pracovisko.STAV.HardwareBunky_OK THEN
		P34_Vizu.IndexStavu_StoperSrobovaniaP3:= 3;
	ELSIF P3_Pracovisko.STAV.Porucha_ST1 THEN
		P34_Vizu.IndexStavu_StoperSrobovaniaP3:= 3;
	ELSIF P3_StoperSrobovania.Automat AND NOT P3_StoperSrobovania.STAV.PoINIT THEN
		P34_Vizu.IndexStavu_StoperSrobovaniaP3:= 1;
	ELSIF P3_StoperSrobovania.Automat AND P3_StoperSrobovania.STAV.PoINIT THEN
		P34_Vizu.IndexStavu_StoperSrobovaniaP3:= 2;
	ELSE
		P34_Vizu.IndexStavu_StoperSrobovaniaP3:= 0;
	END_IF

	//Šrobovanie//
	IF NOT P3_Pracovisko.STAV.HardwareBunky_OK THEN
		P34_Vizu.IndexStavu_SrobovanieP3:= 3;
	ELSIF P3_Pracovisko.STAV.Porucha_ST1 THEN
		P34_Vizu.IndexStavu_SrobovanieP3:= 3;
	ELSIF P3_Srobovanie.Automat AND NOT P3_Srobovanie.STAV.PoINIT THEN
		P34_Vizu.IndexStavu_SrobovanieP3:= 1;
	ELSIF P3_Srobovanie.Automat AND P3_Srobovanie.STAV.PoINIT THEN
		P34_Vizu.IndexStavu_SrobovanieP3:= 2;
	ELSE
		P34_Vizu.IndexStavu_SrobovanieP3:= 0;
	END_IF

	//HV test//
	IF NOT P3_Pracovisko.STAV.HardwareBunky_OK THEN
		P34_Vizu.IndexStavu_HV_Test:= 3;
	ELSIF P3_Pracovisko.STAV.Porucha_ST2 THEN
		P34_Vizu.IndexStavu_HV_Test:= 3;
	ELSIF P3_HV_Test.Automat AND NOT P3_HV_Test.STAV.PoINIT THEN
		P34_Vizu.IndexStavu_HV_Test:= 1;
	ELSIF P3_HV_Test.Automat AND P3_HV_Test.STAV.PoINIT THEN
		P34_Vizu.IndexStavu_HV_Test:= 2;
	ELSE
		P34_Vizu.IndexStavu_HV_Test:= 0;
	END_IF

	//Zdvižka pred Leakage testom A//
	IF P3_Pracovisko.STAV.Porucha_ST3 THEN
		P34_Vizu.IndexStavu_ZdvizkPredLeakTestomA:= 3;
	ELSIF P3_ZdvizkaPredLeakTestA.Automat AND NOT P3_ZdvizkaPredLeakTestA.STAV.PoINIT THEN
		P34_Vizu.IndexStavu_ZdvizkPredLeakTestomA:= 1;
	ELSIF P3_ZdvizkaPredLeakTestA.Automat AND P3_ZdvizkaPredLeakTestA.STAV.PoINIT THEN
		P34_Vizu.IndexStavu_ZdvizkPredLeakTestomA:= 2;
	ELSE
		P34_Vizu.IndexStavu_ZdvizkPredLeakTestomA:= 0;
	END_IF

	//Zdvižka pred Leakage testom B//
	IF P3_Pracovisko.STAV.Porucha_ST4 THEN
		P34_Vizu.IndexStavu_ZdvizkPredLeakTestomB:= 3;
	ELSIF P3_ZdvizkaPredLeakTestB.Automat AND NOT P3_ZdvizkaPredLeakTestB.STAV.PoINIT THEN
		P34_Vizu.IndexStavu_ZdvizkPredLeakTestomB:= 1;
	ELSIF P3_ZdvizkaPredLeakTestB.Automat AND P3_ZdvizkaPredLeakTestB.STAV.PoINIT THEN
		P34_Vizu.IndexStavu_ZdvizkPredLeakTestomB:= 2;
	ELSE
		P34_Vizu.IndexStavu_ZdvizkPredLeakTestomB:= 0;
	END_IF

	//Stoper Leakage Test A//
	IF P3_Pracovisko.STAV.Porucha_ST5 THEN
		P34_Vizu.IndexStavu_StoperLeakageTestA:= 3;
	ELSIF P3_LeakageTestA.Automat AND NOT P3_LeakageTestA.STAV.PoINIT THEN
		P34_Vizu.IndexStavu_StoperLeakageTestA:= 1;
	ELSIF P3_LeakageTestA.Automat AND P3_LeakageTestA.STAV.PoINIT THEN
		P34_Vizu.IndexStavu_StoperLeakageTestA:= 2;
	ELSE
		P34_Vizu.IndexStavu_StoperLeakageTestA:= 0;
	END_IF

	//Stoper Leakage Test B//
	IF P3_Pracovisko.STAV.Porucha_ST6 THEN
		P34_Vizu.IndexStavu_StoperLeakageTestB:= 3;
	ELSIF P3_LeakageTestB.Automat AND NOT P3_LeakageTestB.STAV.PoINIT THEN
		P34_Vizu.IndexStavu_StoperLeakageTestB:= 1;
	ELSIF P3_LeakageTestB.Automat AND P3_LeakageTestB.STAV.PoINIT THEN
		P34_Vizu.IndexStavu_StoperLeakageTestB:= 2;
	ELSE
		P34_Vizu.IndexStavu_StoperLeakageTestB:= 0;
	END_IF

	//Zdvižka za Leakage testom A//
	IF P3_Pracovisko.STAV.Porucha_ST7 THEN
		P34_Vizu.IndexStavu_ZdvizkaZaLeakTestomA:= 3;
	ELSIF P3_ZdvizkaZaLeakTestA.Automat AND NOT P3_ZdvizkaZaLeakTestA.STAV.PoINIT THEN
		P34_Vizu.IndexStavu_ZdvizkaZaLeakTestomA:= 1;
	ELSIF P3_ZdvizkaZaLeakTestA.Automat AND P3_ZdvizkaZaLeakTestA.STAV.PoINIT THEN
		P34_Vizu.IndexStavu_ZdvizkaZaLeakTestomA:= 2;
	ELSE
		P34_Vizu.IndexStavu_ZdvizkaZaLeakTestomA:= 0;
	END_IF

	//Zdvižka za Leakage testom B//
	IF P3_Pracovisko.STAV.Porucha_ST8 THEN
		P34_Vizu.IndexStavu_ZdvizkaZaLeakTestomB:= 3;
	ELSIF P3_ZdvizkaZaLeakTestB.Automat AND NOT P3_ZdvizkaZaLeakTestB.STAV.PoINIT THEN
		P34_Vizu.IndexStavu_ZdvizkaZaLeakTestomB:= 1;
	ELSIF P3_ZdvizkaZaLeakTestB.Automat AND P3_ZdvizkaZaLeakTestB.STAV.PoINIT THEN
		P34_Vizu.IndexStavu_ZdvizkaZaLeakTestomB:= 2;
	ELSE
		P34_Vizu.IndexStavu_ZdvizkaZaLeakTestomB:= 0;
	END_IF

	//*************************************************BUNKA 4**********************************************************//

	//**************Zmeny farieb tlačítok ovládania zámkov bunky 4*********************//
	//Predné dvere //
	IF P4_Pracovisko.OUT.PredneDvere_ZAMKNI AND P4_Pracovisko.IN.PredneDvere_PritomnostAdaptera THEN
		P34_Vizu.TL_PrednyZamok_Farba_P4:= "Button_Green";
	ELSIF P4_Pracovisko.IN.PredneDvere_PritomnostAdaptera THEN
		IF Blikac1s THEN
			P34_Vizu.TL_PrednyZamok_Farba_P4:= "Button_Blue";
		ELSE
			P34_Vizu.TL_PrednyZamok_Farba_P4:= "Operate";
		END_IF
	ELSE
		P34_Vizu.TL_PrednyZamok_Farba_P4:= "Button_Red";
	END_IF

	//Zadné dvere//
	IF P4_Pracovisko.OUT.ZadneDvere_ZAMKNI AND P4_Pracovisko.IN.ZadneDvere_PritomnostAdaptera THEN
		P34_Vizu.TL_ZadnyZamok_Farba_P4:= "Button_Green";
	ELSIF P4_Pracovisko.IN.ZadneDvere_PritomnostAdaptera THEN
		IF Blikac1s THEN
			P34_Vizu.TL_ZadnyZamok_Farba_P4:= "Button_Blue";
		ELSE
			P34_Vizu.TL_ZadnyZamok_Farba_P4:= "Operate";
		END_IF
	ELSE
		P34_Vizu.TL_ZadnyZamok_Farba_P4:= "Button_Red";
	END_IF

	//*****************Zobrazenie warningov bunky 4****************************//
	//0 - Pracovisko je vypnuté.
	//1 - Prebieha inicializácia pracoviska.
	//2 - Na pracovisku prebieha výroba.
	//3 - Prebieha ukončenie pracovného cyklu pracoviska.
	//4 - Prebieha režim vyprázdnenia linky.
	//5 - Niesu založené správne kontakty na Funkčnom teste stanica A !!!
	//6 - Niesu založené správne kontakty na Funkčnom teste stanica B !!!

	IF Linka.PAR.ZvolenyModel = '4F' AND NOT P4_FunkcnyTestA.IN.TypSpodnychKontaktov_4F THEN
		P34_Vizu.WarningsP4_Index:= 5;
	ELSIF Linka.PAR.ZvolenyModel = '5F' AND NOT P4_FunkcnyTestA.IN.TypSpodnychKontaktov_5F_5H THEN
		P34_Vizu.WarningsP4_Index:= 5;
	ELSIF Linka.PAR.ZvolenyModel = '5H' AND NOT P4_FunkcnyTestA.IN.TypSpodnychKontaktov_5F_5H THEN
		P34_Vizu.WarningsP4_Index:= 5;
	ELSIF Linka.PAR.ZvolenyModel = '4F' AND NOT P4_FunkcnyTestB.IN.TypSpodnychKontaktov_4F THEN
		P34_Vizu.WarningsP4_Index:= 6;
	ELSIF Linka.PAR.ZvolenyModel = '5F' AND NOT P4_FunkcnyTestB.IN.TypSpodnychKontaktov_5F_5H THEN
		P34_Vizu.WarningsP4_Index:= 6;
	ELSIF Linka.PAR.ZvolenyModel = '5H' AND NOT P4_FunkcnyTestB.IN.TypSpodnychKontaktov_5F_5H THEN
		P34_Vizu.WarningsP4_Index:= 6;
	ELSIF P4_Pracovisko.STAV.Automat AND NOT P4_Pracovisko.STAV.PoINIT AND NOT P4_Pracovisko.STAV.UkoncenieCyklu_BUSY THEN
		P34_Vizu.WarningsP4_Index:= 1;
	ELSIF Linka.PAR.TestovaciKus THEN
		P34_Vizu.WarningsP4_Index:= 8;
	ELSIF Linka.PAR.VyprazdnenieLinky THEN
		P34_Vizu.WarningsP4_Index:= 4;
	ELSIF P4_Pracovisko.STAV.PoINIT AND NOT P4_Pracovisko.STAV.UkoncenieCyklu_BUSY THEN
		P34_Vizu.WarningsP4_Index:= 2;
	ELSIF P4_Pracovisko.STAV.UkoncenieCyklu_BUSY THEN
		P34_Vizu.WarningsP4_Index:= 3;
	ELSIF NOT P4_Pracovisko.STAV.Automat THEN
		P34_Vizu.WarningsP4_Index:= 0;
	END_IF

	//****************Prepínanie farby textového pola warning bunky 4************************//
	IF P34_Vizu.WarningsP4_Index = 0 THEN
		P34_Vizu.WarningsP4_Farba:= "TextOutput_Grey";
	ELSIF P34_Vizu.WarningsP4_Index = 1 THEN
		P34_Vizu.WarningsP4_Farba:= "TextOutput_Blue";
	ELSIF P34_Vizu.WarningsP4_Index = 2 THEN
		P34_Vizu.WarningsP4_Farba:= "TextOutput_Green";
	ELSIF P34_Vizu.WarningsP4_Index = 3 THEN
		P34_Vizu.WarningsP4_Farba:= "TextOutput_Blue";
	ELSIF P34_Vizu.WarningsP4_Index = 4 THEN
		P34_Vizu.WarningsP4_Farba:= "TextOutput_Green";
	ELSIF P34_Vizu.WarningsP4_Index = 8 THEN
		P34_Vizu.WarningsP4_Farba:= "TextOutput_Green";
	ELSE
		IF Blikac1s THEN
			P34_Vizu.WarningsP4_Farba:= "TextOutput_Orange";
		ELSE
			P34_Vizu.WarningsP4_Farba:= "TextOutput_Grey";
		END_IF
	END_IF

	//*************Zamknutie tlačítok bunky 4************************//
	//Zamknutie tlačítok ovládania zámkov//
	IF P4_Pracovisko.STAV.Automat THEN
		P34_Vizu.TL_OvladaniaZamkov_ENABLE_P4:= FALSE;
	ELSIF P4_FunkcnyTestA.STAV.RR_SekvenciaTestera_BUSY THEN
		P34_Vizu.TL_OvladaniaZamkov_ENABLE_P4:= FALSE;
	ELSIF P4_FunkcnyTestB.STAV.RR_SekvenciaTestera_BUSY THEN
		P34_Vizu.TL_OvladaniaZamkov_ENABLE_P4:= FALSE;
	ELSIF P4_Etiketovacka.STAV.RR_SekvenciaEtiketovania_BUSY THEN
		P34_Vizu.TL_OvladaniaZamkov_ENABLE_P4:= FALSE;
	ELSE
		P34_Vizu.TL_OvladaniaZamkov_ENABLE_P4:= TRUE;
	END_IF

	//Tlačítko Štat Automat//
	IF P4_Pracovisko.STAV.UkoncenieCyklu_BUSY THEN
		P34_Vizu.TL_StartAutomat_ENABLE_P4:= FALSE;
	ELSIF P4_Pracovisko.STAV.PORUCHA THEN
		P34_Vizu.TL_StartAutomat_ENABLE_P4:= FALSE;
	ELSIF NOT Safety.STAV.P4_ZonaBunky_AKTIVNA THEN
		P34_Vizu.TL_StartAutomat_ENABLE_P4:= FALSE;
	ELSIF NOT P4_Pracovisko.STAV.HardwareBunky_OK THEN
		P34_Vizu.TL_StartAutomat_ENABLE_P4:= FALSE;
	ELSE
		P34_Vizu.TL_StartAutomat_ENABLE_P4:= TRUE;
	END_IF

	//Tlačítko Ukončenie Cyklu//
	IF P4_Pracovisko.STAV.PoINIT THEN
		P34_Vizu.TL_KoniecCyklu_ENABLE_P4:= TRUE;
	ELSE
		P34_Vizu.TL_KoniecCyklu_ENABLE_P4:= FALSE;
	END_IF

	//Tlačítko STOP//
	IF P4_Pracovisko.STAV.PoINIT AND NOT P4_Pracovisko.STAV.UkoncenieCyklu_BUSY THEN
		P34_Vizu.TL_STOP_ENABLE_P4:= FALSE;
	ELSE
		P34_Vizu.TL_STOP_ENABLE_P4:= TRUE;
	END_IF

	//Tlačítko Režim Manual//
	IF P4_Pracovisko.STAV.Automat THEN
		P34_Vizu.TL_RezimManual_ENABLE_P4:= FALSE;
	ELSIF NOT P4_Pracovisko.STAV.HardwareBunky_OK THEN
		P34_Vizu.TL_RezimManual_ENABLE_P4:= FALSE;
	ELSE
		P34_Vizu.TL_RezimManual_ENABLE_P4:= TRUE;
	END_IF

	//Tlačítka vypnutia final testov//
//	IF P4_Pracovisko.STAV.Automat THEN
//		P34_Vizu.VolbaFunkcnehoTestu_ENABLE:= FALSE;
//	ELSE
		P34_Vizu.VolbaFunkcnehoTestu_ENABLE:= TRUE;
//	END_IF

	//RR - Ovládanie Funkčného testu A//
	IF P4_FunkcnyTestA.STAV.RR_SekvenciaTestera_BUSY THEN
		P34_Vizu.TL_OvladaniaFunkcTestuA_ENABLE:= FALSE;
	ELSIF NOT Safety.STAV.P4_ZonaBunky_AKTIVNA THEN
		P34_Vizu.TL_OvladaniaFunkcTestuA_ENABLE:= FALSE;
	ELSIF NOT Safety.STAV.Linka_ZonaCS_AKTIVNA THEN
		P34_Vizu.TL_OvladaniaFunkcTestuA_ENABLE:= FALSE;
	ELSE
		P34_Vizu.TL_OvladaniaFunkcTestuA_ENABLE:= TRUE;
	END_IF

	//RR - Ovládanie sekvencie Funkčného Testu A//
	IF NOT Safety.STAV.P4_ZonaBunky_AKTIVNA THEN
		P34_Vizu.TL_SekvencieFunkcTestuA_ENABLE:= FALSE;
	ELSIF NOT Safety.STAV.Linka_ZonaCS_AKTIVNA THEN
		P34_Vizu.TL_SekvencieFunkcTestuA_ENABLE:= FALSE;
	ELSIF NOT P4_FunkcnyTestA.RFID_hlava.PritomnostPaletky THEN
		P34_Vizu.TL_SekvencieFunkcTestuA_ENABLE:= FALSE;
	ELSE
		P34_Vizu.TL_SekvencieFunkcTestuA_ENABLE:= TRUE;
	END_IF

	//RR - Ovládanie Funkčného testu B//
	IF P4_FunkcnyTestB.STAV.RR_SekvenciaTestera_BUSY THEN
		P34_Vizu.TL_OvladaniaFunkcTestuB_ENABLE:= FALSE;
	ELSIF NOT Safety.STAV.P4_ZonaBunky_AKTIVNA THEN
		P34_Vizu.TL_OvladaniaFunkcTestuB_ENABLE:= FALSE;
	ELSIF NOT Safety.STAV.Linka_ZonaCS_AKTIVNA THEN
		P34_Vizu.TL_OvladaniaFunkcTestuB_ENABLE:= FALSE;
	ELSE
		P34_Vizu.TL_OvladaniaFunkcTestuB_ENABLE:= TRUE;
	END_IF

	//RR - Ovládanie sekvencie Funkčného Testu B//
	IF NOT Safety.STAV.P4_ZonaBunky_AKTIVNA THEN
		P34_Vizu.TL_SekvencieFunkcTestuB_ENABLE:= FALSE;
	ELSIF NOT Safety.STAV.Linka_ZonaCS_AKTIVNA THEN
		P34_Vizu.TL_SekvencieFunkcTestuB_ENABLE:= FALSE;
	ELSIF NOT P4_FunkcnyTestB.RFID_hlava.PritomnostPaletky THEN
		P34_Vizu.TL_SekvencieFunkcTestuB_ENABLE:= FALSE;
	ELSE
		P34_Vizu.TL_SekvencieFunkcTestuB_ENABLE:= TRUE;
	END_IF

	//RR - Ovládanie etiketovania//
	IF P4_Etiketovacka.STAV.RR_SekvenciaEtiketovania_BUSY THEN
		P34_Vizu.TL_OvladaniaEtiketovania_ENABLE:= FALSE;
	ELSIF NOT Safety.STAV.P4_ZonaBunky_AKTIVNA THEN
		P34_Vizu.TL_OvladaniaEtiketovania_ENABLE:= FALSE;
	ELSIF NOT Safety.STAV.Linka_ZonaCS_AKTIVNA THEN
		P34_Vizu.TL_OvladaniaEtiketovania_ENABLE:= FALSE;
	ELSE
		P34_Vizu.TL_OvladaniaEtiketovania_ENABLE:= TRUE;
	END_IF

	//RR - Ovládanie sekvencie etiketovania//
	IF NOT Safety.STAV.P4_ZonaBunky_AKTIVNA THEN
		P34_Vizu.TL_SekvencieEtiketovania_ENABLE:= FALSE;
	ELSIF NOT Safety.STAV.Linka_ZonaCS_AKTIVNA THEN
		P34_Vizu.TL_SekvencieEtiketovania_ENABLE:= FALSE;
	ELSIF P4_Etiketovacka.STAV.RR_SekvenciaEtiketovania_BUSY THEN
		P34_Vizu.TL_SekvencieEtiketovania_ENABLE:= FALSE;
	ELSIF P4_Etiketovacka.ServoZdvihuAplikatora.Status.ActPosition > 5 THEN
		P34_Vizu.TL_SekvencieEtiketovania_ENABLE:= FALSE;
	ELSIF NOT P4_Etiketovacka.RFID_hlava.PritomnostPaletky THEN
		P34_Vizu.TL_SekvencieEtiketovania_ENABLE:= FALSE;
	ELSIF NOT P4_Etiketovacka.IN.Aplikator_OtocenyVZAD THEN
		P34_Vizu.TL_SekvencieEtiketovania_ENABLE:= FALSE;
	ELSIF NOT P4_Etiketovacka.IN.Aplikator_ZASUNUTY THEN
		P34_Vizu.TL_SekvencieEtiketovania_ENABLE:= FALSE;
	ELSE
		P34_Vizu.TL_SekvencieEtiketovania_ENABLE:= TRUE;
	END_IF

	//RR - Tlačítka ovládania zdvihu aplikátora//
	IF NOT Safety.STAV.P4_ZonaBunky_AKTIVNA THEN
		P34_Vizu.TL_ZdvihAplikEtiketovania_ENABLE:= FALSE;
	ELSE
		P34_Vizu.TL_ZdvihAplikEtiketovania_ENABLE:= TRUE;
	END_IF

	//RR - Tlačítko výtah čítanie paletky//
	IF P4_Vytah.RFID_hlava.PritomnostPaletky THEN
		P34_Vizu.Vytah_CitaniePaletky_ENABLE:= TRUE;
	ELSE
		P34_Vizu.Vytah_CitaniePaletky_ENABLE:= FALSE;
	END_IF

	//RR - Tlačítko výťah zápis paletky//
	IF P4_Vytah.RFID_hlava.PritomnostPaletky THEN
		P34_Vizu.Vytah_ZapisPaletky_ENABLE:= TRUE;
	ELSE
		P34_Vizu.Vytah_ZapisPaletky_ENABLE:= FALSE;
	END_IF

	//************Prepínanie stavov pracovísk - Bunka 4**************************//
	//Dopravníky//
	IF P4_Dopravniky.Automat AND NOT P4_Dopravniky.STAV.PoINIT THEN
		P34_Vizu.IndexStavu_DopravnikP4:= 1;
	ELSIF P4_Dopravniky.Automat AND P4_Dopravniky.STAV.PoINIT THEN
		P34_Vizu.IndexStavu_DopravnikP4:= 2;
	ELSE
		P34_Vizu.IndexStavu_DopravnikP4:= 0;
	END_IF

	//Spodný stoper//
	IF P4_SpodnyStoper.Automat AND NOT P4_SpodnyStoper.STAV.PoINIT THEN
		P34_Vizu.IndexStavu_SpodnyStoperP4:= 1;
	ELSIF P4_SpodnyStoper.Automat AND P4_SpodnyStoper.STAV.PoINIT THEN
		P34_Vizu.IndexStavu_SpodnyStoperP4:= 2;
	ELSE
		P34_Vizu.IndexStavu_SpodnyStoperP4:= 0;
	END_IF

	//Stoper Funkčný Test A//
	IF P4_Pracovisko.STAV.Porucha_ST1 THEN
		P34_Vizu.IndexStavu_StoperFunkcnyTestA:= 3;
	ELSIF P4_FunkcnyTestA.Automat AND NOT P4_FunkcnyTestA.STAV.PoINIT THEN
		P34_Vizu.IndexStavu_StoperFunkcnyTestA:= 1;
	ELSIF P4_FunkcnyTestA.Automat AND P4_FunkcnyTestA.STAV.PoINIT THEN
		P34_Vizu.IndexStavu_StoperFunkcnyTestA:= 2;
	ELSE
		P34_Vizu.IndexStavu_StoperFunkcnyTestA:= 0;
	END_IF

	//Stoper Funkčný Test B//
	IF P4_Pracovisko.STAV.Porucha_ST2 THEN
		P34_Vizu.IndexStavu_StoperFunkcnyTestB:= 3;
	ELSIF P4_FunkcnyTestB.Automat AND NOT P4_FunkcnyTestB.STAV.PoINIT THEN
		P34_Vizu.IndexStavu_StoperFunkcnyTestB:= 1;
	ELSIF P4_FunkcnyTestB.Automat AND P4_FunkcnyTestB.STAV.PoINIT THEN
		P34_Vizu.IndexStavu_StoperFunkcnyTestB:= 2;
	ELSE
		P34_Vizu.IndexStavu_StoperFunkcnyTestB:= 0;
	END_IF

	//Zdvižka za Funkčným testom A//
	IF P4_Pracovisko.STAV.Porucha_ST3 THEN
		P34_Vizu.IndexStavu_ZdvizkaZaFunkTestomA:= 3;
	ELSIF P4_ZdvizkaZaFunkcTestA.Automat AND NOT P4_ZdvizkaZaFunkcTestA.STAV.PoINIT THEN
		P34_Vizu.IndexStavu_ZdvizkaZaFunkTestomA:= 1;
	ELSIF P4_ZdvizkaZaFunkcTestA.Automat AND P4_ZdvizkaZaFunkcTestA.STAV.PoINIT THEN
		P34_Vizu.IndexStavu_ZdvizkaZaFunkTestomA:= 2;
	ELSE
		P34_Vizu.IndexStavu_ZdvizkaZaFunkTestomA:= 0;
	END_IF

	//Zdvižka za Funkčným testom B//
	IF P4_Pracovisko.STAV.Porucha_ST4 THEN
		P34_Vizu.IndexStavu_ZdvizkaZaFunkTestomB:= 3;
	ELSIF P4_ZdvizkaZaFunkcTestB.Automat AND NOT P4_ZdvizkaZaFunkcTestB.STAV.PoINIT THEN
		P34_Vizu.IndexStavu_ZdvizkaZaFunkTestomB:= 1;
	ELSIF P4_ZdvizkaZaFunkcTestB.Automat AND P4_ZdvizkaZaFunkcTestB.STAV.PoINIT THEN
		P34_Vizu.IndexStavu_ZdvizkaZaFunkTestomB:= 2;
	ELSE
		P34_Vizu.IndexStavu_ZdvizkaZaFunkTestomB:= 0;
	END_IF

	//Stoper Etiketovačky//
	IF NOT P4_Pracovisko.STAV.HardwareBunky_OK THEN
		P34_Vizu.IndexStavu_StoperEtiketovackyP4:= 3;
	ELSIF P4_Pracovisko.STAV.Porucha_ST5 THEN
		P34_Vizu.IndexStavu_StoperEtiketovackyP4:= 3;
	ELSIF P4_Etiketovacka.Automat AND NOT P4_Etiketovacka.STAV.PoINIT THEN
		P34_Vizu.IndexStavu_StoperEtiketovackyP4:= 1;
	ELSIF P4_Etiketovacka.Automat AND P4_Etiketovacka.STAV.PoINIT THEN
		P34_Vizu.IndexStavu_StoperEtiketovackyP4:= 2;
	ELSE
		P34_Vizu.IndexStavu_StoperEtiketovackyP4:= 0;
	END_IF

	//Výťah//
	IF NOT P4_Pracovisko.STAV.HardwareVytahu_OK THEN
		P34_Vizu.IndexStavu_Vytah:= 3;
	ELSIF P4_Pracovisko.STAV.Porucha_ST6 THEN
		P34_Vizu.IndexStavu_Vytah:= 3;
	ELSIF P4_Vytah.Automat AND NOT P4_Vytah.STAV.PoINIT THEN
		P34_Vizu.IndexStavu_Vytah:= 1;
	ELSIF P4_Vytah.Automat AND P4_Vytah.STAV.PoINIT THEN
		P34_Vizu.IndexStavu_Vytah:= 2;
	ELSE
		P34_Vizu.IndexStavu_Vytah:= 0;
	END_IF

		END_PROGRAM

PROGRAM _EXIT
		(* Insert code here *)

		END_PROGRAM
```

### Program Logical/Program/Pracovisko_4/P4_OvladSafety (IEC)

#### Main.st - Init, cyclic, exit code
```iecst
PROGRAM _INIT
	(* Insert code here *)

END_PROGRAM

PROGRAM _CYCLIC

	//******************************************Ovládanie zámkov dverí bunky****************************************//
	//Predné dvere //
	IF P34_Vizu.TL_ZamkniPrednyZamok_P4 THEN
		IF NOT P4_Pracovisko.OUT.PredneDvere_ZAMKNI AND P4_Pracovisko.IN.PredneDvere_PritomnostAdaptera THEN
			P4_Pracovisko.OUT.PredneDvere_ZAMKNI:= TRUE;
		ELSIF P4_Pracovisko.OUT.PredneDvere_ZAMKNI THEN
			P4_Pracovisko.OUT.PredneDvere_ZAMKNI:= FALSE;
		END_IF
		P34_Vizu.TL_ZamkniPrednyZamok_P4:= FALSE;
	END_IF

	//Zadné dvere//
	IF P34_Vizu.TL_ZamkniZadnyZamok_P4 THEN
		IF NOT P4_Pracovisko.OUT.ZadneDvere_ZAMKNI AND P4_Pracovisko.IN.ZadneDvere_PritomnostAdaptera THEN
			P4_Pracovisko.OUT.ZadneDvere_ZAMKNI:= TRUE;
		ELSIF P4_Pracovisko.OUT.ZadneDvere_ZAMKNI THEN
			P4_Pracovisko.OUT.ZadneDvere_ZAMKNI:= FALSE;
		END_IF
		P34_Vizu.TL_ZamkniZadnyZamok_P4:= FALSE;
	END_IF

	//******************************************Reset zóny výtahu*********************************************//
	IF Safety.STAV.Linka_ZonaCS_AKTIVNA AND
		(Safety.STAV.P4_Vytah_Bariera_AKTIVNA OR Safety.STAV.P4_Vytah_Muting_AKTIVNY) AND
		NOT Safety.STAV.P4_ZonaVytahu_AKTIVNA THEN
		Safety.OUT.P4_ResetZonyVytahu:= TRUE;
	ELSE
		Safety.OUT.P4_ResetZonyVytahu:= FALSE;
	END_IF

	//*****************************************Reset zóny bunky************************************************//
	IF Safety.STAV.Linka_ZonaCS_AKTIVNA AND
		(Safety.STAV.P4_Bunka_Zamky_AKTIVNE OR Safety.STAV.P4_VyblokovanieZamkov_AKTIVNE) AND
		NOT Safety.STAV.P4_ZonaBunky_AKTIVNA AND
		(Safety.STAV.P4_Bunka_VstupBariera_AKTIVNA OR Safety.STAV.P3_Bunka_Zamky_AKTIVNE)AND
		(Safety.STAV.P4_VystupBunky_VstupBar_AKTIVNA OR Safety.STAV.P4_VystupBunky_VystupBar_AKTIVNA) THEN
		Safety.OUT.P4_ResetZonyBunky:= TRUE;
	ELSE
		Safety.OUT.P4_ResetZonyBunky:= FALSE;
	END_IF

END_PROGRAM

PROGRAM _EXIT
	(* Insert code here *)

END_PROGRAM
```

### Program Logical/Program/Pracovisko_4/P4_Mapping_IO (IEC)
